LIN {X 0,Y 390.118,Z 490.981,A -85,B 0,C 180,E1 -11473.897,E2 -11473.897} C_VEL
LIN {X 0,Y 390.11,Z 491.016,A -85,B 0,C 180,E1 -11476.798,E2 -11476.798} C_VEL
LIN {X 0,Y 390.064,Z 491.01,A -85,B 0,C 180,E1 -11479.562,E2 -11479.562} C_VEL
LIN {X 0,Y 390.038,Z 491.022,A -85,B 0,C 180,E1 -11482.449,E2 -11482.449} C_VEL
LIN {X 0,Y 390.06,Z 491.021,A -85,B 0,C 180,E1 -11486.045,E2 -11486.045} C_VEL
LIN {X 0,Y 390.038,Z 491.013,A -85,B 0,C 180,E1 -11488.498,E2 -11488.498} C_VEL
LIN {X 0,Y 390.109,Z 491.015,A -85,B 0,C 180,E1 -11492.07,E2 -11492.07} C_VEL
LIN {X 0,Y 390.071,Z 491.003,A -85,B 0,C 180,E1 -11495.519,E2 -11495.519} C_VEL
LIN {X 0,Y 390.054,Z 491.022,A -85,B 0,C 180,E1 -11498.878,E2 -11498.878} C_VEL
LIN {X 0,Y 390.119,Z 490.998,A -85,B 0,C 180,E1 -11502.167,E2 -11502.167} C_VEL
LIN {X 0,Y 390.135,Z 491.009,A -85,B 0,C 180,E1 -11505.393,E2 -11505.393} C_VEL
LIN {X 0,Y 390.139,Z 490.999,A -85,B 0,C 180,E1 -11508.571,E2 -11508.571} C_VEL
LIN {X 0,Y 390.298,Z 490.981,A -85,B 0,C 180,E1 -11512.033,E2 -11512.033} C_VEL
LIN {X 0,Y 390.225,Z 490.997,A -85,B 0,C 180,E1 -11514.834,E2 -11514.834} C_VEL
LIN {X 0,Y 390.412,Z 490.954,A -85,B 0,C 180,E1 -11517.937,E2 -11517.937} C_VEL
LIN {X 0,Y 390.541,Z 490.951,A -85,B 0,C 180,E1 -11520,E2 -11520} C_VEL
LIN {X 0,Y 390.308,Z 490.984,A -85,B 0,C 180,E1 -11523.097,E2 -11523.097} C_VEL
LIN {X 0,Y 390.32,Z 490.966,A -85,B 0,C 180,E1 -11526.202,E2 -11526.202} C_VEL
LIN {X 0,Y 390.197,Z 491.003,A -85,B 0,C 180,E1 -11529.329,E2 -11529.329} C_VEL
LIN {X 0,Y 390.187,Z 490.982,A -85,B 0,C 180,E1 -11533.439,E2 -11533.439} C_VEL
LIN {X 0,Y 390.142,Z 491.01,A -85,B 0,C 180,E1 -11537.308,E2 -11537.308} C_VEL
LIN {X 0,Y 390.081,Z 491.003,A -85,B 0,C 180,E1 -11540.471,E2 -11540.471} C_VEL
LIN {X 0,Y 390.072,Z 491.023,A -85,B 0,C 180,E1 -11544.482,E2 -11544.482} C_VEL
LIN {X 0,Y 390.112,Z 491.001,A -85,B 0,C 180,E1 -11547.931,E2 -11547.931} C_VEL
LIN {X 0,Y 390.018,Z 491.022,A -85,B 0,C 180,E1 -11551.505,E2 -11551.505} C_VEL
LIN {X 0,Y 390.081,Z 491.019,A -85,B 0,C 180,E1 -11555.208,E2 -11555.208} C_VEL
LIN {X 0,Y 390.091,Z 491.019,A -85,B 0,C 180,E1 -11559.093,E2 -11559.093} C_VEL
LIN {X 0,Y 390.077,Z 491.015,A -85,B 0,C 180,E1 -11562.381,E2 -11562.381} C_VEL
LIN {X 0,Y 390.054,Z 491.005,A -85,B 0,C 180,E1 -11566.115,E2 -11566.115} C_VEL
LIN {X 0,Y 390.055,Z 491.022,A -85,B 0,C 180,E1 -11569.562,E2 -11569.562} C_VEL
LIN {X 0,Y 390.042,Z 490.971,A -85,B 0,C 180,E1 -11572.45,E2 -11572.45} C_VEL
LIN {X 0,Y 390.067,Z 491.009,A -85,B 0,C 180,E1 -11575.976,E2 -11575.976} C_VEL
LIN {X 0,Y 390.107,Z 491.228,A -85,B 0,C 180,E1 -11577.132,E2 -11577.132} C_VEL
LIN {X 0,Y 392.197,Z 500.873,A -85,B 0,C 180,E1 -11579.885,E2 -11579.885} C_VEL
LIN {X 0,Y 394.038,Z 510.309,A -85,B 0,C 180,E1 -11582.373,E2 -11582.373} C_VEL
LIN {X 0,Y 394.142,Z 513.122,A -85,B 0,C 180,E1 -11583.07,E2 -11583.07} C_VEL
LIN {X 0,Y 393.369,Z 521.493,A -85,B 0,C 180,E1 -11585.111,E2 -11585.111} C_VEL
LIN {X 0,Y 394.757,Z 528.148,A -85,B 0,C 180,E1 -11585.38,E2 -11585.38} C_VEL
LIN {X 0,Y 400.375,Z 555.374,A -85,B 0,C 180,E1 -11586.267,E2 -11586.267} C_VEL
LIN {X 0,Y 400.741,Z 558.243,A -85,B 0,C 180,E1 -11586.345,E2 -11586.345} C_VEL
LIN {X 0,Y 398.955,Z 657.044,A -85,B 0,C 180,E1 -11588.153,E2 -11588.153} C_VEL
LIN {X 0,Y 398.444,Z 667.994,A -85,B 0,C 180,E1 -11588.463,E2 -11588.463} C_VEL
LIN {X 0,Y 397.788,Z 678.984,A -85,B 0,C 180,E1 -11588.902,E2 -11588.902} C_VEL
LIN {X 0,Y 397.102,Z 688.994,A -85,B 0,C 180,E1 -11589.42,E2 -11589.42} C_VEL
LIN {X 0,Y 396.287,Z 698.786,A -85,B 0,C 180,E1 -11590.042,E2 -11590.042} C_VEL
LIN {X 0,Y 395.442,Z 708.675,A -85,B 0,C 180,E1 -11590.805,E2 -11590.805} C_VEL
LIN {X 0,Y 394.447,Z 718.401,A -85,B 0,C 180,E1 -11591.698,E2 -11591.698} C_VEL
LIN {X 0,Y 393.41,Z 727.821,A -85,B 0,C 180,E1 -11592.723,E2 -11592.723} C_VEL
LIN {X 0,Y 392.435,Z 736.845,A -85,B 0,C 180,E1 -11593.884,E2 -11593.884} C_VEL
LIN {X 0,Y 391.671,Z 743.822,A -85,B 0,C 180,E1 -11594.919,E2 -11594.919} C_VEL
LIN {X 0,Y 390.934,Z 750.826,A -85,B 0,C 180,E1 -11596.117,E2 -11596.117} C_VEL
LIN {X 0,Y 390.32,Z 757.827,A -85,B 0,C 180,E1 -11597.522,E2 -11597.522} C_VEL
LIN {X 0,Y 389.661,Z 764.367,A -85,B 0,C 180,E1 -11599.084,E2 -11599.084} C_VEL
LIN {X 0,Y 389.23,Z 769.8,A -85,B 0,C 180,E1 -11600.648,E2 -11600.648} C_VEL
LIN {X 0,Y 388.923,Z 774.244,A -85,B 0,C 180,E1 -11602.211,E2 -11602.211} C_VEL
LIN {X 0,Y 388.775,Z 777.942,A -85,B 0,C 180,E1 -11603.856,E2 -11603.856} C_VEL
LIN {X 0,Y 388.707,Z 779.727,A -85,B 0,C 180,E1 -11604.813,E2 -11604.813} C_VEL
LIN {X 0,Y 388.63,Z 782.408,A -85,B 0,C 180,E1 -11606.89,E2 -11606.89} C_VEL
LIN {X 0,Y 388.702,Z 783.698,A -85,B 0,C 180,E1 -11608.964,E2 -11608.964} C_VEL
LIN {X 0,Y 388.707,Z 783.95,A -85,B 0,C 180,E1 -11610,E2 -11610} C_VEL
LIN {X 0,Y 388.659,Z 783.225,A -85,B 0,C 180,E1 -11612.073,E2 -11612.073} C_VEL
LIN {X 0,Y 388.63,Z 782.408,A -85,B 0,C 180,E1 -11613.11,E2 -11613.11} C_VEL
LIN {X 0,Y 388.704,Z 779.727,A -85,B 0,C 180,E1 -11615.187,E2 -11615.187} C_VEL
LIN {X 0,Y 388.845,Z 776.773,A -85,B 0,C 180,E1 -11616.747,E2 -11616.747} C_VEL
LIN {X 0,Y 389.002,Z 772.946,A -85,B 0,C 180,E1 -11618.31,E2 -11618.31} C_VEL
LIN {X 0,Y 389.339,Z 768.184,A -85,B 0,C 180,E1 -11619.874,E2 -11619.874} C_VEL
LIN {X 0,Y 389.993,Z 761.241,A -85,B 0,C 180,E1 -11621.697,E2 -11621.697} C_VEL
LIN {X 0,Y 390.661,Z 754.026,A -85,B 0,C 180,E1 -11623.26,E2 -11623.26} C_VEL
LIN {X 0,Y 391.34,Z 746.947,A -85,B 0,C 180,E1 -11624.561,E2 -11624.561} C_VEL
LIN {X 0,Y 392.036,Z 740.483,A -85,B 0,C 180,E1 -11625.599,E2 -11625.599} C_VEL
LIN {X 0,Y 393.053,Z 731,A -85,B 0,C 180,E1 -11626.891,E2 -11626.891} C_VEL
LIN {X 0,Y 394.065,Z 722.123,A -85,B 0,C 180,E1 -11627.917,E2 -11627.917} C_VEL
LIN {X 0,Y 395.042,Z 713.07,A -85,B 0,C 180,E1 -11628.811,E2 -11628.811} C_VEL
LIN {X 0,Y 396.028,Z 702.261,A -85,B 0,C 180,E1 -11629.705,E2 -11629.705} C_VEL
LIN {X 0,Y 396.826,Z 692.523,A -85,B 0,C 180,E1 -11630.373,E2 -11630.373} C_VEL
LIN {X 0,Y 397.585,Z 681.704,A -85,B 0,C 180,E1 -11630.974,E2 -11630.974} C_VEL
LIN {X 0,Y 398.346,Z 669.818,A -85,B 0,C 180,E1 -11631.474,E2 -11631.474} C_VEL
LIN {X 0,Y 398.878,Z 658.403,A -85,B 0,C 180,E1 -11631.817,E2 -11631.817} C_VEL
LIN {X 0,Y 399.554,Z 628.292,A -85,B 0,C 180,E1 -11632.39,E2 -11632.39} C_VEL
LIN {X 0,Y 400.705,Z 557.213,A -85,B 0,C 180,E1 -11633.677,E2 -11633.677} C_VEL
LIN {X 0,Y 394.872,Z 528.424,A -85,B 0,C 180,E1 -11634.607,E2 -11634.607} C_VEL
LIN {X 0,Y 393.382,Z 521.582,A -85,B 0,C 180,E1 -11634.877,E2 -11634.877} C_VEL
LIN {X 0,Y 394.231,Z 512.042,A -85,B 0,C 180,E1 -11637.195,E2 -11637.195} C_VEL
LIN {X 0,Y 392.995,Z 504.589,A -85,B 0,C 180,E1 -11639.163,E2 -11639.163} C_VEL
LIN {X 0,Y 390.582,Z 493.387,A -85,B 0,C 180,E1 -11642.252,E2 -11642.252} C_VEL
LIN {X 0,Y 390.082,Z 491.039,A -85,B 0,C 180,E1 -11643.005,E2 -11643.005} C_VEL
LIN {X 0,Y 390.055,Z 490.963,A -85,B 0,C 180,E1 -11646.483,E2 -11646.483} C_VEL
LIN {X 0,Y 390.069,Z 491.006,A -85,B 0,C 180,E1 -11649.218,E2 -11649.218} C_VEL
LIN {X 0,Y 390.042,Z 491.009,A -85,B 0,C 180,E1 -11652.374,E2 -11652.374} C_VEL
LIN {X 0,Y 390.042,Z 491.021,A -85,B 0,C 180,E1 -11655.354,E2 -11655.354} C_VEL
LIN {X 0,Y 390.065,Z 491.014,A -85,B 0,C 180,E1 -11658.191,E2 -11658.191} C_VEL
LIN {X 0,Y 390.091,Z 491.018,A -85,B 0,C 180,E1 -11660.907,E2 -11660.907} C_VEL
LIN {X 0,Y 390.081,Z 491.019,A -85,B 0,C 180,E1 -11664.792,E2 -11664.792} C_VEL
LIN {X 0,Y 390.018,Z 491.022,A -85,B 0,C 180,E1 -11668.495,E2 -11668.495} C_VEL
LIN {X 0,Y 390.112,Z 491.001,A -85,B 0,C 180,E1 -11672.069,E2 -11672.069} C_VEL
LIN {X 0,Y 390.072,Z 491.023,A -85,B 0,C 180,E1 -11675.518,E2 -11675.518} C_VEL
LIN {X 0,Y 390.081,Z 491.003,A -85,B 0,C 180,E1 -11679.529,E2 -11679.529} C_VEL
LIN {X 0,Y 390.131,Z 491.015,A -85,B 0,C 180,E1 -11683.247,E2 -11683.247} C_VEL
LIN {X 0,Y 390.187,Z 490.982,A -85,B 0,C 180,E1 -11686.561,E2 -11686.561} C_VEL
LIN {X 0,Y 390.197,Z 491.003,A -85,B 0,C 180,E1 -11690.671,E2 -11690.671} C_VEL
LIN {X 0,Y 390.32,Z 490.966,A -85,B 0,C 180,E1 -11693.798,E2 -11693.798} C_VEL
LIN {X 0,Y 390.412,Z 490.976,A -85,B 0,C 180,E1 -11697.936,E2 -11697.936} C_VEL
LIN {X 0,Y 390.541,Z 490.951,A -85,B 0,C 180,E1 -11700,E2 -11700} C_VEL
LIN {X 0,Y 390.308,Z 490.97,A -85,B 0,C 180,E1 -11703.096,E2 -11703.096} C_VEL
LIN {X 0,Y 390.293,Z 490.989,A -85,B 0,C 180,E1 -11706.649,E2 -11706.649} C_VEL
LIN {X 0,Y 390.196,Z 490.986,A -85,B 0,C 180,E1 -11709.328,E2 -11709.328} C_VEL
LIN {X 0,Y 390.186,Z 491.008,A -85,B 0,C 180,E1 -11713.438,E2 -11713.438} C_VEL
LIN {X 0,Y 390.14,Z 490.994,A -85,B 0,C 180,E1 -11717.307,E2 -11717.307} C_VEL
LIN {X 0,Y 390.079,Z 491.017,A -85,B 0,C 180,E1 -11720.47,E2 -11720.47} C_VEL
LIN {X 0,Y 390.08,Z 491.008,A -85,B 0,C 180,E1 -11723.351,E2 -11723.351} C_VEL
LIN {X 0,Y 390.105,Z 491.013,A -85,B 0,C 180,E1 -11726.768,E2 -11726.768} C_VEL
LIN {X 0,Y 390.036,Z 491.009,A -85,B 0,C 180,E1 -11730.299,E2 -11730.299} C_VEL
LIN {X 0,Y 390.047,Z 491.021,A -85,B 0,C 180,E1 -11732.72,E2 -11732.72} C_VEL
LIN {X 0,Y 390.049,Z 491.013,A -85,B 0,C 180,E1 -11735.826,E2 -11735.826} C_VEL
LIN {X 0,Y 390.064,Z 491.022,A -85,B 0,C 180,E1 -11739.219,E2 -11739.219} C_VEL
LIN {X 0,Y 390.114,Z 491.015,A -85,B 0,C 180,E1 -11742.387,E2 -11742.387} C_VEL
LIN {X 0,Y 390.11,Z 490.994,A -85,B 0,C 180,E1 -11745.365,E2 -11745.365} C_VEL
LIN {X 0,Y 390.098,Z 490.993,A -85,B 0,C 180,E1 -11748.197,E2 -11748.197} C_VEL
LIN {X 0,Y 390.09,Z 491.018,A -85,B 0,C 180,E1 -11750.909,E2 -11750.909} C_VEL
LIN {X 0,Y 390.079,Z 491.013,A -85,B 0,C 180,E1 -11754.793,E2 -11754.793} C_VEL
LIN {X 0,Y 390.028,Z 491.03,A -85,B 0,C 180,E1 -11757.875,E2 -11757.875} C_VEL
LIN {X 0,Y 390.06,Z 491.023,A -85,B 0,C 180,E1 -11760.891,E2 -11760.891} C_VEL
LIN {X 0,Y 390.106,Z 491.018,A -85,B 0,C 180,E1 -11764.382,E2 -11764.382} C_VEL
LIN {X 0,Y 390.035,Z 491.028,A -85,B 0,C 180,E1 -11767.766,E2 -11767.766} C_VEL
LIN {X 0,Y 390.101,Z 491.019,A -85,B 0,C 180,E1 -11771.078,E2 -11771.078} C_VEL
LIN {X 0,Y 390.135,Z 491.015,A -85,B 0,C 180,E1 -11774.323,E2 -11774.323} C_VEL
LIN {X 0,Y 390.167,Z 491.011,A -85,B 0,C 180,E1 -11777.517,E2 -11777.517} C_VEL
LIN {X 0,Y 390.241,Z 491.299,A -85,B 0,C 180,E1 -11780.378,E2 -11780.378} C_VEL
LIN {X 0,Y 390.604,Z 492.537,A -85,B 0,C 180,E1 -11781.137,E2 -11781.137} C_VEL
LIN {X 0,Y 392.054,Z 494.823,A -85,B 0,C 180,E1 -11782.457,E2 -11782.457} C_VEL
LIN {X 0,Y 393.897,Z 496.346,A -85,B 0,C 180,E1 -11784.369,E2 -11784.369} C_VEL
LIN {X 0,Y 395.019,Z 496.962,A -85,B 0,C 180,E1 -11785.919,E2 -11785.919} C_VEL
LIN {X 0,Y 395.996,Z 497.339,A -85,B 0,C 180,E1 -11787.966,E2 -11787.966} C_VEL
LIN {X 0,Y 396.223,Z 497.592,A -85,B 0,C 180,E1 -11788.984,E2 -11788.984} C_VEL
LIN {X 0,Y 396.324,Z 497.476,A -85,B 0,C 180,E1 -11790,E2 -11790} C_VEL
LIN {X 0,Y 396.113,Z 497.471,A -85,B 0,C 180,E1 -11791.525,E2 -11791.525} C_VEL
LIN {X 0,Y 395.594,Z 497.134,A -85,B 0,C 180,E1 -11793.055,E2 -11793.055} C_VEL
LIN {X 0,Y 394.296,Z 496.586,A -85,B 0,C 180,E1 -11795.113,E2 -11795.113} C_VEL
LIN {X 0,Y 392.392,Z 495.186,A -85,B 0,C 180,E1 -11797.202,E2 -11797.202} C_VEL
LIN {X 0,Y 390.757,Z 492.871,A -85,B 0,C 180,E1 -11798.717,E2 -11798.717} C_VEL
LIN {X 0,Y 390.301,Z 491.64,A -85,B 0,C 180,E1 -11799.326,E2 -11799.326} C_VEL
LIN {X 0,Y 390.165,Z 491.041,A -85,B 0,C 180,E1 -11800.377,E2 -11800.377} C_VEL
LIN {X 0,Y 390.165,Z 491.011,A -85,B 0,C 180,E1 -11803.542,E2 -11803.542} C_VEL
LIN {X 0,Y 390.144,Z 491.014,A -85,B 0,C 180,E1 -11807.307,E2 -11807.307} C_VEL
LIN {X 0,Y 390.082,Z 491.022,A -85,B 0,C 180,E1 -11810.47,E2 -11810.47} C_VEL
LIN {X 0,Y 390.084,Z 491.021,A -85,B 0,C 180,E1 -11813.351,E2 -11813.351} C_VEL
LIN {X 0,Y 390.108,Z 491.018,A -85,B 0,C 180,E1 -11816.768,E2 -11816.768} C_VEL
LIN {X 0,Y 390.038,Z 491.028,A -85,B 0,C 180,E1 -11820.299,E2 -11820.299} C_VEL
LIN {X 0,Y 390.01,Z 491.028,A -85,B 0,C 180,E1 -11820.819,E2 -11820.819} C_VEL
LIN {X 0,Y 389.336,Z 491.114,A -85,B 0,C 180,E1 -11821.681,E2 -11821.681} C_VEL
LIN {X 0,Y 386.486,Z 491.468,A -85,B 0,C 180,E1 -11823.083,E2 -11823.083} C_VEL
LIN {X 0,Y 384.087,Z 491.769,A -85,B 0,C 180,E1 -11824.216,E2 -11824.216} C_VEL
LIN {X 0,Y 383.069,Z 491.887,A -85,B 0,C 180,E1 -11825.092,E2 -11825.092} C_VEL
LIN {X 0,Y 382.993,Z 491.887,A -85,B 0,C 180,E1 -11825.388,E2 -11825.388} C_VEL
LIN {X 0,Y 383.003,Z 491.896,A -85,B 0,C 180,E1 -11828.6,E2 -11828.6} C_VEL
LIN {X 0,Y 383.04,Z 491.882,A -85,B 0,C 180,E1 -11831.339,E2 -11831.339} C_VEL
LIN {X 0,Y 383.061,Z 491.865,A -85,B 0,C 180,E1 -11834.314,E2 -11834.314} C_VEL
LIN {X 0,Y 383.068,Z 491.892,A -85,B 0,C 180,E1 -11837.249,E2 -11837.249} C_VEL
LIN {X 0,Y 383.012,Z 491.898,A -85,B 0,C 180,E1 -11840.412,E2 -11840.412} C_VEL
LIN {X 0,Y 383.018,Z 491.888,A -85,B 0,C 180,E1 -11844.044,E2 -11844.044} C_VEL
LIN {X 0,Y 383.028,Z 491.897,A -85,B 0,C 180,E1 -11847.853,E2 -11847.853} C_VEL
LIN {X 0,Y 383.055,Z 491.891,A -85,B 0,C 180,E1 -11851.72,E2 -11851.72} C_VEL
LIN {X 0,Y 383.043,Z 491.879,A -85,B 0,C 180,E1 -11855.04,E2 -11855.04} C_VEL
LIN {X 0,Y 382.99,Z 491.904,A -85,B 0,C 180,E1 -11858.469,E2 -11858.469} C_VEL
LIN {X 0,Y 383.08,Z 491.877,A -85,B 0,C 180,E1 -11861.828,E2 -11861.828} C_VEL
LIN {X 0,Y 383.101,Z 491.886,A -85,B 0,C 180,E1 -11865.118,E2 -11865.118} C_VEL
LIN {X 0,Y 383.089,Z 491.88,A -85,B 0,C 180,E1 -11868.358,E2 -11868.358} C_VEL
LIN {X 0,Y 383.255,Z 491.858,A -85,B 0,C 180,E1 -11871.976,E2 -11871.976} C_VEL
LIN {X 0,Y 383.197,Z 491.873,A -85,B 0,C 180,E1 -11874.739,E2 -11874.739} C_VEL
LIN {X 0,Y 383.38,Z 491.829,A -85,B 0,C 180,E1 -11877.899,E2 -11877.899} C_VEL
LIN {X 0,Y 383.511,Z 491.827,A -85,B 0,C 180,E1 -11880,E2 -11880} C_VEL
LIN {X 0,Y 383.244,Z 491.863,A -85,B 0,C 180,E1 -11883.154,E2 -11883.154} C_VEL
LIN {X 0,Y 383.277,Z 491.844,A -85,B 0,C 180,E1 -11886.317,E2 -11886.317} C_VEL
LIN {X 0,Y 383.144,Z 491.881,A -85,B 0,C 180,E1 -11889.503,E2 -11889.503} C_VEL
LIN {X 0,Y 383.118,Z 491.862,A -85,B 0,C 180,E1 -11893.537,E2 -11893.537} C_VEL
LIN {X 0,Y 383.088,Z 491.888,A -85,B 0,C 180,E1 -11897.455,E2 -11897.455} C_VEL
LIN {X 0,Y 383.022,Z 491.881,A -85,B 0,C 180,E1 -11900.647,E2 -11900.647} C_VEL
LIN {X 0,Y 383.02,Z 491.897,A -85,B 0,C 180,E1 -11903.809,E2 -11903.809} C_VEL
LIN {X 0,Y 383.074,Z 491.884,A -85,B 0,C 180,E1 -11906.124,E2 -11906.124} C_VEL
LIN {X 0,Y 382.986,Z 491.901,A -85,B 0,C 180,E1 -11909.701,E2 -11909.701} C_VEL
LIN {X 0,Y 382.998,Z 491.89,A -85,B 0,C 180,E1 -11913.402,E2 -11913.402} C_VEL
LIN {X 0,Y 383.029,Z 491.898,A -85,B 0,C 180,E1 -11916.166,E2 -11916.166} C_VEL
LIN {X 0,Y 383.016,Z 491.9,A -85,B 0,C 180,E1 -11919.958,E2 -11919.958} C_VEL
LIN {X 0,Y 383.029,Z 491.896,A -85,B 0,C 180,E1 -11922.784,E2 -11922.784} C_VEL
LIN {X 0,Y 382.996,Z 491.887,A -85,B 0,C 180,E1 -11925.79,E2 -11925.79} C_VEL
LIN {X 0,Y 382.987,Z 491.902,A -85,B 0,C 180,E1 -11928.797,E2 -11928.797} C_VEL
LIN {X 0,Y 382.998,Z 491.852,A -85,B 0,C 180,E1 -11932.097,E2 -11932.097} C_VEL
LIN {X 0,Y 383.017,Z 491.864,A -85,B 0,C 180,E1 -11935.333,E2 -11935.333} C_VEL
LIN {X 0,Y 383.077,Z 492.078,A -85,B 0,C 180,E1 -11936.728,E2 -11936.728} C_VEL
LIN {X 0,Y 385.189,Z 501.84,A -85,B 0,C 180,E1 -11939.582,E2 -11939.582} C_VEL
LIN {X 0,Y 387.187,Z 512.271,A -85,B 0,C 180,E1 -11942.383,E2 -11942.383} C_VEL
LIN {X 0,Y 386.939,Z 516.944,A -85,B 0,C 180,E1 -11943.578,E2 -11943.578} C_VEL
LIN {X 0,Y 386.564,Z 521.303,A -85,B 0,C 180,E1 -11944.645,E2 -11944.645} C_VEL
LIN {X 0,Y 388.306,Z 529.362,A -85,B 0,C 180,E1 -11944.971,E2 -11944.971} C_VEL
LIN {X 0,Y 394.047,Z 557.41,A -85,B 0,C 180,E1 -11945.906,E2 -11945.906} C_VEL
LIN {X 0,Y 393.732,Z 585.51,A -85,B 0,C 180,E1 -11946.433,E2 -11946.433} C_VEL
LIN {X 0,Y 392.374,Z 656.846,A -85,B 0,C 180,E1 -11947.767,E2 -11947.767} C_VEL
LIN {X 0,Y 391.856,Z 667.796,A -85,B 0,C 180,E1 -11948.083,E2 -11948.083} C_VEL
LIN {X 0,Y 391.176,Z 678.786,A -85,B 0,C 180,E1 -11948.527,E2 -11948.527} C_VEL
LIN {X 0,Y 390.448,Z 688.583,A -85,B 0,C 180,E1 -11949.039,E2 -11949.039} C_VEL
LIN {X 0,Y 389.575,Z 698.907,A -85,B 0,C 180,E1 -11949.708,E2 -11949.708} C_VEL
LIN {X 0,Y 388.729,Z 708.52,A -85,B 0,C 180,E1 -11950.464,E2 -11950.464} C_VEL
LIN {X 0,Y 387.702,Z 718.202,A -85,B 0,C 180,E1 -11951.368,E2 -11951.368} C_VEL
LIN {X 0,Y 386.601,Z 727.622,A -85,B 0,C 180,E1 -11952.409,E2 -11952.409} C_VEL
LIN {X 0,Y 385.56,Z 736.645,A -85,B 0,C 180,E1 -11953.589,E2 -11953.589} C_VEL
LIN {X 0,Y 384.758,Z 743.622,A -85,B 0,C 180,E1 -11954.642,E2 -11954.642} C_VEL
LIN {X 0,Y 383.905,Z 751.284,A -85,B 0,C 180,E1 -11955.99,E2 -11955.99} C_VEL
LIN {X 0,Y 383.234,Z 758.766,A -85,B 0,C 180,E1 -11957.557,E2 -11957.557} C_VEL
LIN {X 0,Y 382.637,Z 764.167,A -85,B 0,C 180,E1 -11958.881,E2 -11958.881} C_VEL
LIN {X 0,Y 382.165,Z 769.6,A -85,B 0,C 180,E1 -11960.473,E2 -11960.473} C_VEL
LIN {X 0,Y 381.851,Z 774.045,A -85,B 0,C 180,E1 -11962.066,E2 -11962.066} C_VEL
LIN {X 0,Y 381.71,Z 777.59,A -85,B 0,C 180,E1 -11963.658,E2 -11963.658} C_VEL
LIN {X 0,Y 381.616,Z 779.528,A -85,B 0,C 180,E1 -11964.717,E2 -11964.717} C_VEL
LIN {X 0,Y 381.541,Z 782.21,A -85,B 0,C 180,E1 -11966.832,E2 -11966.832} C_VEL
LIN {X 0,Y 381.616,Z 783.5,A -85,B 0,C 180,E1 -11968.945,E2 -11968.945} C_VEL
LIN {X 0,Y 381.638,Z 783.753,A -85,B 0,C 180,E1 -11970,E2 -11970} C_VEL
LIN {X 0,Y 381.558,Z 783.027,A -85,B 0,C 180,E1 -11972.111,E2 -11972.111} C_VEL
LIN {X 0,Y 381.541,Z 782.21,A -85,B 0,C 180,E1 -11973.168,E2 -11973.168} C_VEL
LIN {X 0,Y 381.615,Z 779.528,A -85,B 0,C 180,E1 -11975.283,E2 -11975.283} C_VEL
LIN {X 0,Y 381.757,Z 776.574,A -85,B 0,C 180,E1 -11976.872,E2 -11976.872} C_VEL
LIN {X 0,Y 381.95,Z 772.747,A -85,B 0,C 180,E1 -11978.465,E2 -11978.465} C_VEL
LIN {X 0,Y 382.301,Z 767.985,A -85,B 0,C 180,E1 -11980.058,E2 -11980.058} C_VEL
LIN {X 0,Y 382.974,Z 761.041,A -85,B 0,C 180,E1 -11981.914,E2 -11981.914} C_VEL
LIN {X 0,Y 383.555,Z 755.164,A -85,B 0,C 180,E1 -11983.24,E2 -11983.24} C_VEL
LIN {X 0,Y 384.429,Z 746.748,A -85,B 0,C 180,E1 -11984.829,E2 -11984.829} C_VEL
LIN {X 0,Y 385.167,Z 740.284,A -85,B 0,C 180,E1 -11985.884,E2 -11985.884} C_VEL
LIN {X 0,Y 386.213,Z 730.801,A -85,B 0,C 180,E1 -11987.199,E2 -11987.199} C_VEL
LIN {X 0,Y 387.287,Z 721.924,A -85,B 0,C 180,E1 -11988.242,E2 -11988.242} C_VEL
LIN {X 0,Y 388.305,Z 712.871,A -85,B 0,C 180,E1 -11989.15,E2 -11989.15} C_VEL
LIN {X 0,Y 389.329,Z 702.062,A -85,B 0,C 180,E1 -11990.058,E2 -11990.058} C_VEL
LIN {X 0,Y 390.264,Z 691.158,A -85,B 0,C 180,E1 -11990.806,E2 -11990.806} C_VEL
LIN {X 0,Y 391.058,Z 680.146,A -85,B 0,C 180,E1 -11991.41,E2 -11991.41} C_VEL
LIN {X 0,Y 391.808,Z 668.708,A -85,B 0,C 180,E1 -11991.885,E2 -11991.885} C_VEL
LIN {X 0,Y 392.303,Z 658.205,A -85,B 0,C 180,E1 -11992.202,E2 -11992.202} C_VEL
LIN {X 0,Y 393.006,Z 628.094,A -85,B 0,C 180,E1 -11992.784,E2 -11992.784} C_VEL
LIN {X 0,Y 394.133,Z 557.774,A -85,B 0,C 180,E1 -11994.082,E2 -11994.082} C_VEL
LIN {X 0,Y 388.314,Z 529.209,A -85,B 0,C 180,E1 -11995.032,E2 -11995.032} C_VEL
LIN {X 0,Y 386.58,Z 521.374,A -85,B 0,C 180,E1 -11995.345,E2 -11995.345} C_VEL
LIN {X 0,Y 387.295,Z 513.75,A -85,B 0,C 180,E1 -11997.23,E2 -11997.23} C_VEL
LIN {X 0,Y 386.212,Z 506.655,A -85,B 0,C 180,E1 -11999.135,E2 -11999.135} C_VEL
LIN {X 0,Y 383.975,Z 496.243,A -85,B 0,C 180,E1 -12002.058,E2 -12002.058} C_VEL
LIN {X 0,Y 383.069,Z 491.935,A -85,B 0,C 180,E1 -12003.363,E2 -12003.363} C_VEL
LIN {X 0,Y 383.03,Z 491.837,A -85,B 0,C 180,E1 -12006.164,E2 -12006.164} C_VEL
LIN {X 0,Y 383.007,Z 491.9,A -85,B 0,C 180,E1 -12009.957,E2 -12009.957} C_VEL
LIN {X 0,Y 383.003,Z 491.881,A -85,B 0,C 180,E1 -12012.778,E2 -12012.778} C_VEL
LIN {X 0,Y 382.995,Z 491.903,A -85,B 0,C 180,E1 -12015.788,E2 -12015.788} C_VEL
LIN {X 0,Y 383.011,Z 491.894,A -85,B 0,C 180,E1 -12018.79,E2 -12018.79} C_VEL
LIN {X 0,Y 382.999,Z 491.892,A -85,B 0,C 180,E1 -12022.095,E2 -12022.095} C_VEL
LIN {X 0,Y 383.014,Z 491.896,A -85,B 0,C 180,E1 -12025.331,E2 -12025.331} C_VEL
LIN {X 0,Y 382.977,Z 491.903,A -85,B 0,C 180,E1 -12029.081,E2 -12029.081} C_VEL
LIN {X 0,Y 383.051,Z 491.879,A -85,B 0,C 180,E1 -12032.697,E2 -12032.697} C_VEL
LIN {X 0,Y 383.045,Z 491.892,A -85,B 0,C 180,E1 -12035.039,E2 -12035.039} C_VEL
LIN {X 0,Y 382.985,Z 491.89,A -85,B 0,C 180,E1 -12038.468,E2 -12038.468} C_VEL
LIN {X 0,Y 383.082,Z 491.891,A -85,B 0,C 180,E1 -12041.827,E2 -12041.827} C_VEL
LIN {X 0,Y 383.102,Z 491.877,A -85,B 0,C 180,E1 -12045.118,E2 -12045.118} C_VEL
LIN {X 0,Y 383.09,Z 491.883,A -85,B 0,C 180,E1 -12048.357,E2 -12048.357} C_VEL
LIN {X 0,Y 383.257,Z 491.862,A -85,B 0,C 180,E1 -12051.974,E2 -12051.974} C_VEL
LIN {X 0,Y 383.191,Z 491.853,A -85,B 0,C 180,E1 -12054.738,E2 -12054.738} C_VEL
LIN {X 0,Y 383.38,Z 491.852,A -85,B 0,C 180,E1 -12057.898,E2 -12057.898} C_VEL
LIN {X 0,Y 383.511,Z 491.827,A -85,B 0,C 180,E1 -12060,E2 -12060} C_VEL
LIN {X 0,Y 383.244,Z 491.85,A -85,B 0,C 180,E1 -12063.153,E2 -12063.153} C_VEL
LIN {X 0,Y 383.252,Z 491.865,A -85,B 0,C 180,E1 -12066.641,E2 -12066.641} C_VEL
LIN {X 0,Y 383.143,Z 491.863,A -85,B 0,C 180,E1 -12069.502,E2 -12069.502} C_VEL
LIN {X 0,Y 383.117,Z 491.889,A -85,B 0,C 180,E1 -12073.536,E2 -12073.536} C_VEL
LIN {X 0,Y 383.086,Z 491.872,A -85,B 0,C 180,E1 -12077.454,E2 -12077.454} C_VEL
LIN {X 0,Y 383.022,Z 491.896,A -85,B 0,C 180,E1 -12080.648,E2 -12080.648} C_VEL
LIN {X 0,Y 383.024,Z 491.882,A -85,B 0,C 180,E1 -12083.807,E2 -12083.807} C_VEL
LIN {X 0,Y 383.071,Z 491.891,A -85,B 0,C 180,E1 -12086.123,E2 -12086.123} C_VEL
LIN {X 0,Y 383.041,Z 491.892,A -85,B 0,C 180,E1 -12088.492,E2 -12088.492} C_VEL
LIN {X 0,Y 383,Z 491.899,A -85,B 0,C 180,E1 -12092.427,E2 -12092.427} C_VEL
LIN {X 0,Y 383.018,Z 491.888,A -85,B 0,C 180,E1 -12095.956,E2 -12095.956} C_VEL
LIN {X 0,Y 383.012,Z 491.898,A -85,B 0,C 180,E1 -12099.588,E2 -12099.588} C_VEL
LIN {X 0,Y 383.058,Z 491.894,A -85,B 0,C 180,E1 -12102.788,E2 -12102.788} C_VEL
LIN {X 0,Y 383.062,Z 491.863,A -85,B 0,C 180,E1 -12105.8,E2 -12105.8} C_VEL
LIN {X 0,Y 383.038,Z 491.886,A -85,B 0,C 180,E1 -12108.786,E2 -12108.786} C_VEL
LIN {X 0,Y 382.997,Z 491.886,A -85,B 0,C 180,E1 -12112.096,E2 -12112.096} C_VEL
LIN {X 0,Y 383.012,Z 491.898,A -85,B 0,C 180,E1 -12115.332,E2 -12115.332} C_VEL
LIN {X 0,Y 382.981,Z 491.905,A -85,B 0,C 180,E1 -12119.082,E2 -12119.082} C_VEL
LIN {X 0,Y 383.051,Z 491.897,A -85,B 0,C 180,E1 -12122.698,E2 -12122.698} C_VEL
LIN {X 0,Y 383.028,Z 491.9,A -85,B 0,C 180,E1 -12126.193,E2 -12126.193} C_VEL
LIN {X 0,Y 383.05,Z 491.897,A -85,B 0,C 180,E1 -12129.599,E2 -12129.599} C_VEL
LIN {X 0,Y 383.1,Z 491.892,A -85,B 0,C 180,E1 -12132.932,E2 -12132.932} C_VEL
LIN {X 0,Y 383.196,Z 492.132,A -85,B 0,C 180,E1 -12136.59,E2 -12136.59} C_VEL
LIN {X 0,Y 383.443,Z 493.257,A -85,B 0,C 180,E1 -12137.11,E2 -12137.11} C_VEL
LIN {X 0,Y 384.779,Z 495.64,A -85,B 0,C 180,E1 -12137.942,E2 -12137.942} C_VEL
LIN {X 0,Y 386.586,Z 497.173,A -85,B 0,C 180,E1 -12139.019,E2 -12139.019} C_VEL
LIN {X 0,Y 389.002,Z 498.608,A -85,B 0,C 180,E1 -12140.577,E2 -12140.577} C_VEL
LIN {X 0,Y 390.336,Z 500.879,A -85,B 0,C 180,E1 -12141.719,E2 -12141.719} C_VEL
LIN {X 0,Y 391.901,Z 502.624,A -85,B 0,C 180,E1 -12143.177,E2 -12143.177} C_VEL
LIN {X 0,Y 393.414,Z 503.635,A -85,B 0,C 180,E1 -12144.876,E2 -12144.876} C_VEL
LIN {X 0,Y 394.726,Z 504.158,A -85,B 0,C 180,E1 -12146.938,E2 -12146.938} C_VEL
LIN {X 0,Y 395.358,Z 504.638,A -85,B 0,C 180,E1 -12148.981,E2 -12148.981} C_VEL
LIN {X 0,Y 395.358,Z 504.639,A -85,B 0,C 180,E1 -12151.019,E2 -12151.019} C_VEL
LIN {X 0,Y 394.726,Z 504.155,A -85,B 0,C 180,E1 -12153.062,E2 -12153.062} C_VEL
LIN {X 0,Y 393.418,Z 503.612,A -85,B 0,C 180,E1 -12155.124,E2 -12155.124} C_VEL
LIN {X 0,Y 391.495,Z 502.25,A -85,B 0,C 180,E1 -12157.219,E2 -12157.219} C_VEL
LIN {X 0,Y 389.779,Z 500.121,A -85,B 0,C 180,E1 -12158.752,E2 -12158.752} C_VEL
LIN {X 0,Y 388.706,Z 498.318,A -85,B 0,C 180,E1 -12159.627,E2 -12159.627} C_VEL
LIN {X 0,Y 385.613,Z 496.448,A -85,B 0,C 180,E1 -12161.565,E2 -12161.565} C_VEL
LIN {X 0,Y 384.062,Z 494.607,A -85,B 0,C 180,E1 -12162.483,E2 -12162.483} C_VEL
LIN {X 0,Y 383.247,Z 492.572,A -85,B 0,C 180,E1 -12163.135,E2 -12163.135} C_VEL
LIN {X 0,Y 383.122,Z 491.933,A -85,B 0,C 180,E1 -12163.796,E2 -12163.796} C_VEL
LIN {X 0,Y 383.09,Z 491.892,A -85,B 0,C 180,E1 -12167.454,E2 -12167.454} C_VEL
LIN {X 0,Y 383.024,Z 491.902,A -85,B 0,C 180,E1 -12170.647,E2 -12170.647} C_VEL
LIN {X 0,Y 383.028,Z 491.9,A -85,B 0,C 180,E1 -12173.807,E2 -12173.807} C_VEL
LIN {X 0,Y 383.051,Z 491.897,A -85,B 0,C 180,E1 -12177.302,E2 -12177.302} C_VEL
LIN {X 0,Y 382.981,Z 491.905,A -85,B 0,C 180,E1 -12180.918,E2 -12180.918} C_VEL
LIN {X 0,Y 383.012,Z 491.898,A -85,B 0,C 180,E1 -12184.668,E2 -12184.668} C_VEL
LIN {X 0,Y 382.993,Z 491.887,A -85,B 0,C 180,E1 -12185.388,E2 -12185.388} C_VEL
LIN {X 0,Y 382.35,Z 491.964,A -85,B 0,C 180,E1 -12186.266,E2 -12186.266} C_VEL
LIN {X 0,Y 379.533,Z 492.33,A -85,B 0,C 180,E1 -12187.694,E2 -12187.694} C_VEL
LIN {X 0,Y 377.128,Z 492.641,A -85,B 0,C 180,E1 -12188.848,E2 -12188.848} C_VEL
LIN {X 0,Y 376.082,Z 492.77,A -85,B 0,C 180,E1 -12189.74,E2 -12189.74} C_VEL
LIN {X 0,Y 375.99,Z 492.777,A -85,B 0,C 180,E1 -12190.043,E2 -12190.043} C_VEL
LIN {X 0,Y 375.991,Z 492.737,A -85,B 0,C 180,E1 -12193.756,E2 -12193.756} C_VEL
LIN {X 0,Y 375.992,Z 492.775,A -85,B 0,C 180,E1 -12196.8,E2 -12196.8} C_VEL
LIN {X 0,Y 375.988,Z 492.767,A -85,B 0,C 180,E1 -12200.028,E2 -12200.028} C_VEL
LIN {X 0,Y 375.957,Z 492.769,A -85,B 0,C 180,E1 -12203.495,E2 -12203.495} C_VEL
LIN {X 0,Y 375.953,Z 492.777,A -85,B 0,C 180,E1 -12205.889,E2 -12205.889} C_VEL
LIN {X 0,Y 375.961,Z 492.761,A -85,B 0,C 180,E1 -12209.688,E2 -12209.688} C_VEL
LIN {X 0,Y 375.994,Z 492.774,A -85,B 0,C 180,E1 -12212.142,E2 -12212.142} C_VEL
LIN {X 0,Y 375.997,Z 492.761,A -85,B 0,C 180,E1 -12214.539,E2 -12214.539} C_VEL
LIN {X 0,Y 375.959,Z 492.775,A -85,B 0,C 180,E1 -12218.046,E2 -12218.046} C_VEL
LIN {X 0,Y 376.015,Z 492.76,A -85,B 0,C 180,E1 -12221.474,E2 -12221.474} C_VEL
LIN {X 0,Y 376.049,Z 492.766,A -85,B 0,C 180,E1 -12224.833,E2 -12224.833} C_VEL
LIN {X 0,Y 376.041,Z 492.761,A -85,B 0,C 180,E1 -12228.137,E2 -12228.137} C_VEL
LIN {X 0,Y 376.211,Z 492.735,A -85,B 0,C 180,E1 -12231.919,E2 -12231.919} C_VEL
LIN {X 0,Y 376.169,Z 492.75,A -85,B 0,C 180,E1 -12234.64,E2 -12234.64} C_VEL
LIN {X 0,Y 376.346,Z 492.704,A -85,B 0,C 180,E1 -12237.86,E2 -12237.86} C_VEL
LIN {X 0,Y 376.48,Z 492.702,A -85,B 0,C 180,E1 -12240.001,E2 -12240.001} C_VEL
LIN {X 0,Y 376.183,Z 492.743,A -85,B 0,C 180,E1 -12243.213,E2 -12243.213} C_VEL
LIN {X 0,Y 376.235,Z 492.721,A -85,B 0,C 180,E1 -12246.436,E2 -12246.436} C_VEL
LIN {X 0,Y 376.111,Z 492.758,A -85,B 0,C 180,E1 -12249.682,E2 -12249.682} C_VEL
LIN {X 0,Y 376.082,Z 492.738,A -85,B 0,C 180,E1 -12253.658,E2 -12253.658} C_VEL
LIN {X 0,Y 376.037,Z 492.766,A -85,B 0,C 180,E1 -12257.608,E2 -12257.608} C_VEL
LIN {X 0,Y 375.972,Z 492.759,A -85,B 0,C 180,E1 -12260.833,E2 -12260.833} C_VEL
LIN {X 0,Y 375.984,Z 492.776,A -85,B 0,C 180,E1 -12264.283,E2 -12264.283} C_VEL
LIN {X 0,Y 376.014,Z 492.757,A -85,B 0,C 180,E1 -12266.653,E2 -12266.653} C_VEL
LIN {X 0,Y 375.959,Z 492.779,A -85,B 0,C 180,E1 -12270.314,E2 -12270.314} C_VEL
LIN {X 0,Y 375.955,Z 492.77,A -85,B 0,C 180,E1 -12274.112,E2 -12274.112} C_VEL
LIN {X 0,Y 375.951,Z 492.776,A -85,B 0,C 180,E1 -12276.742,E2 -12276.742} C_VEL
LIN {X 0,Y 375.994,Z 492.774,A -85,B 0,C 180,E1 -12279.973,E2 -12279.973} C_VEL
LIN {X 0,Y 375.936,Z 492.782,A -85,B 0,C 180,E1 -12283.765,E2 -12283.765} C_VEL
LIN {X 0,Y 375.932,Z 492.76,A -85,B 0,C 180,E1 -12286.812,E2 -12286.812} C_VEL
LIN {X 0,Y 375.961,Z 492.766,A -85,B 0,C 180,E1 -12290.538,E2 -12290.538} C_VEL
LIN {X 0,Y 375.962,Z 492.714,A -85,B 0,C 180,E1 -12293.496,E2 -12293.496} C_VEL
LIN {X 0,Y 376.015,Z 492.918,A -85,B 0,C 180,E1 -12296.299,E2 -12296.299} C_VEL
LIN {X 0,Y 377.84,Z 501.257,A -85,B 0,C 180,E1 -12298.829,E2 -12298.829} C_VEL
LIN {X 0,Y 380.078,Z 512.248,A -85,B 0,C 180,E1 -12301.868,E2 -12301.868} C_VEL
LIN {X 0,Y 380.347,Z 515.117,A -85,B 0,C 180,E1 -12302.652,E2 -12302.652} C_VEL
LIN {X 0,Y 379.777,Z 521.222,A -85,B 0,C 180,E1 -12304.173,E2 -12304.173} C_VEL
LIN {X 0,Y 384.822,Z 544.293,A -85,B 0,C 180,E1 -12305.032,E2 -12305.032} C_VEL
LIN {X 0,Y 387.733,Z 559.553,A -85,B 0,C 180,E1 -12305.534,E2 -12305.534} C_VEL
LIN {X 0,Y 385.84,Z 655.308,A -85,B 0,C 180,E1 -12307.335,E2 -12307.335} C_VEL
LIN {X 0,Y 385.325,Z 666.686,A -85,B 0,C 180,E1 -12307.656,E2 -12307.656} C_VEL
LIN {X 0,Y 384.678,Z 677.228,A -85,B 0,C 180,E1 -12308.076,E2 -12308.076} C_VEL
LIN {X 0,Y 383.895,Z 687.416,A -85,B 0,C 180,E1 -12308.6,E2 -12308.6} C_VEL
LIN {X 0,Y 383.08,Z 697.285,A -85,B 0,C 180,E1 -12309.234,E2 -12309.234} C_VEL
LIN {X 0,Y 381.979,Z 708.796,A -85,B 0,C 180,E1 -12310.15,E2 -12310.15} C_VEL
LIN {X 0,Y 380.968,Z 718.004,A -85,B 0,C 180,E1 -12311.026,E2 -12311.026} C_VEL
LIN {X 0,Y 379.77,Z 727.422,A -85,B 0,C 180,E1 -12312.082,E2 -12312.082} C_VEL
LIN {X 0,Y 378.723,Z 736.446,A -85,B 0,C 180,E1 -12313.284,E2 -12313.284} C_VEL
LIN {X 0,Y 377.856,Z 743.422,A -85,B 0,C 180,E1 -12314.354,E2 -12314.354} C_VEL
LIN {X 0,Y 376.878,Z 751.745,A -85,B 0,C 180,E1 -12315.859,E2 -12315.859} C_VEL
LIN {X 0,Y 376.243,Z 758.566,A -85,B 0,C 180,E1 -12317.322,E2 -12317.322} C_VEL
LIN {X 0,Y 375.625,Z 763.968,A -85,B 0,C 180,E1 -12318.67,E2 -12318.67} C_VEL
LIN {X 0,Y 375.117,Z 769.401,A -85,B 0,C 180,E1 -12320.293,E2 -12320.293} C_VEL
LIN {X 0,Y 374.801,Z 773.846,A -85,B 0,C 180,E1 -12321.916,E2 -12321.916} C_VEL
LIN {X 0,Y 374.628,Z 777.391,A -85,B 0,C 180,E1 -12323.537,E2 -12323.537} C_VEL
LIN {X 0,Y 374.53,Z 779.33,A -85,B 0,C 180,E1 -12324.616,E2 -12324.616} C_VEL
LIN {X 0,Y 374.455,Z 782.012,A -85,B 0,C 180,E1 -12326.772,E2 -12326.772} C_VEL
LIN {X 0,Y 374.516,Z 783.302,A -85,B 0,C 180,E1 -12328.925,E2 -12328.925} C_VEL
LIN {X 0,Y 374.553,Z 783.555,A -85,B 0,C 180,E1 -12330,E2 -12330} C_VEL
LIN {X 0,Y 374.457,Z 782.828,A -85,B 0,C 180,E1 -12332.151,E2 -12332.151} C_VEL
LIN {X 0,Y 374.455,Z 782.012,A -85,B 0,C 180,E1 -12333.228,E2 -12333.228} C_VEL
LIN {X 0,Y 374.53,Z 779.33,A -85,B 0,C 180,E1 -12335.384,E2 -12335.384} C_VEL
LIN {X 0,Y 374.677,Z 776.375,A -85,B 0,C 180,E1 -12337.003,E2 -12337.003} C_VEL
LIN {X 0,Y 374.878,Z 772.548,A -85,B 0,C 180,E1 -12338.626,E2 -12338.626} C_VEL
LIN {X 0,Y 375.248,Z 767.785,A -85,B 0,C 180,E1 -12340.249,E2 -12340.249} C_VEL
LIN {X 0,Y 375.984,Z 760.842,A -85,B 0,C 180,E1 -12342.139,E2 -12342.139} C_VEL
LIN {X 0,Y 376.61,Z 754.965,A -85,B 0,C 180,E1 -12343.489,E2 -12343.489} C_VEL
LIN {X 0,Y 377.338,Z 748.112,A -85,B 0,C 180,E1 -12344.838,E2 -12344.838} C_VEL
LIN {X 0,Y 378.282,Z 740.085,A -85,B 0,C 180,E1 -12346.181,E2 -12346.181} C_VEL
LIN {X 0,Y 379.367,Z 730.601,A -85,B 0,C 180,E1 -12347.52,E2 -12347.52} C_VEL
LIN {X 0,Y 380.508,Z 721.724,A -85,B 0,C 180,E1 -12348.578,E2 -12348.578} C_VEL
LIN {X 0,Y 381.685,Z 711.424,A -85,B 0,C 180,E1 -12349.614,E2 -12349.614} C_VEL
LIN {X 0,Y 382.642,Z 701.864,A -85,B 0,C 180,E1 -12350.424,E2 -12350.424} C_VEL
LIN {X 0,Y 383.626,Z 690.96,A -85,B 0,C 180,E1 -12351.183,E2 -12351.183} C_VEL
LIN {X 0,Y 384.445,Z 679.948,A -85,B 0,C 180,E1 -12351.797,E2 -12351.797} C_VEL
LIN {X 0,Y 385.189,Z 669.422,A -85,B 0,C 180,E1 -12352.246,E2 -12352.246} C_VEL
LIN {X 0,Y 385.743,Z 658.007,A -85,B 0,C 180,E1 -12352.601,E2 -12352.601} C_VEL
LIN {X 0,Y 386.48,Z 627.896,A -85,B 0,C 180,E1 -12353.191,E2 -12353.191} C_VEL
LIN {X 0,Y 387.65,Z 558.758,A -85,B 0,C 180,E1 -12354.487,E2 -12354.487} C_VEL
LIN {X 0,Y 382.041,Z 531.207,A -85,B 0,C 180,E1 -12355.427,E2 -12355.427} C_VEL
LIN {X 0,Y 379.807,Z 521.353,A -85,B 0,C 180,E1 -12355.813,E2 -12355.813} C_VEL
LIN {X 0,Y 379.969,Z 518.94,A -85,B 0,C 180,E1 -12356.353,E2 -12356.353} C_VEL
LIN {X 0,Y 380.357,Z 514.5,A -85,B 0,C 180,E1 -12357.511,E2 -12357.511} C_VEL
LIN {X 0,Y 379.019,Z 506.787,A -85,B 0,C 180,E1 -12359.65,E2 -12359.65} C_VEL
LIN {X 0,Y 376.598,Z 495.581,A -85,B 0,C 180,E1 -12362.883,E2 -12362.883} C_VEL
LIN {X 0,Y 376.016,Z 492.796,A -85,B 0,C 180,E1 -12363.782,E2 -12363.782} C_VEL
LIN {X 0,Y 375.952,Z 492.716,A -85,B 0,C 180,E1 -12366.74,E2 -12366.74} C_VEL
LIN {X 0,Y 375.987,Z 492.774,A -85,B 0,C 180,E1 -12369.97,E2 -12369.97} C_VEL
LIN {X 0,Y 375.928,Z 492.761,A -85,B 0,C 180,E1 -12373.765,E2 -12373.765} C_VEL
LIN {X 0,Y 375.957,Z 492.772,A -85,B 0,C 180,E1 -12377.703,E2 -12377.703} C_VEL
LIN {X 0,Y 375.965,Z 492.777,A -85,B 0,C 180,E1 -12380.537,E2 -12380.537} C_VEL
LIN {X 0,Y 375.961,Z 492.778,A -85,B 0,C 180,E1 -12383.494,E2 -12383.494} C_VEL
LIN {X 0,Y 375.955,Z 492.77,A -85,B 0,C 180,E1 -12385.888,E2 -12385.888} C_VEL
LIN {X 0,Y 375.959,Z 492.779,A -85,B 0,C 180,E1 -12389.686,E2 -12389.686} C_VEL
LIN {X 0,Y 376.014,Z 492.757,A -85,B 0,C 180,E1 -12393.347,E2 -12393.347} C_VEL
LIN {X 0,Y 375.977,Z 492.776,A -85,B 0,C 180,E1 -12396.887,E2 -12396.887} C_VEL
LIN {X 0,Y 375.991,Z 492.762,A -85,B 0,C 180,E1 -12400.339,E2 -12400.339} C_VEL
LIN {X 0,Y 376.021,Z 492.768,A -85,B 0,C 180,E1 -12403.718,E2 -12403.718} C_VEL
LIN {X 0,Y 376.096,Z 492.738,A -85,B 0,C 180,E1 -12407.041,E2 -12407.041} C_VEL
LIN {X 0,Y 376.111,Z 492.758,A -85,B 0,C 180,E1 -12410.318,E2 -12410.318} C_VEL
LIN {X 0,Y 376.235,Z 492.721,A -85,B 0,C 180,E1 -12413.564,E2 -12413.564} C_VEL
LIN {X 0,Y 376.346,Z 492.729,A -85,B 0,C 180,E1 -12417.859,E2 -12417.859} C_VEL
LIN {X 0,Y 376.48,Z 492.702,A -85,B 0,C 180,E1 -12419.999,E2 -12419.999} C_VEL
LIN {X 0,Y 376.182,Z 492.73,A -85,B 0,C 180,E1 -12423.212,E2 -12423.212} C_VEL
LIN {X 0,Y 376.217,Z 492.741,A -85,B 0,C 180,E1 -12426.63,E2 -12426.63} C_VEL
LIN {X 0,Y 376.111,Z 492.737,A -85,B 0,C 180,E1 -12429.681,E2 -12429.681} C_VEL
LIN {X 0,Y 376.081,Z 492.766,A -85,B 0,C 180,E1 -12433.657,E2 -12433.657} C_VEL
LIN {X 0,Y 376.035,Z 492.75,A -85,B 0,C 180,E1 -12437.607,E2 -12437.607} C_VEL
LIN {X 0,Y 375.97,Z 492.775,A -85,B 0,C 180,E1 -12440.832,E2 -12440.832} C_VEL
LIN {X 0,Y 375.985,Z 492.756,A -85,B 0,C 180,E1 -12444.281,E2 -12444.281} C_VEL
LIN {X 0,Y 376.011,Z 492.769,A -85,B 0,C 180,E1 -12446.652,E2 -12446.652} C_VEL
LIN {X 0,Y 375.968,Z 492.774,A -85,B 0,C 180,E1 -12449.079,E2 -12449.079} C_VEL
LIN {X 0,Y 375.948,Z 492.778,A -85,B 0,C 180,E1 -12452.828,E2 -12452.828} C_VEL
LIN {X 0,Y 375.95,Z 492.771,A -85,B 0,C 180,E1 -12455.416,E2 -12455.416} C_VEL
LIN {X 0,Y 375.968,Z 492.778,A -85,B 0,C 180,E1 -12458.271,E2 -12458.271} C_VEL
LIN {X 0,Y 375.981,Z 492.768,A -85,B 0,C 180,E1 -12461.61,E2 -12461.61} C_VEL
LIN {X 0,Y 376.008,Z 492.751,A -85,B 0,C 180,E1 -12465.255,E2 -12465.255} C_VEL
LIN {X 0,Y 375.994,Z 492.767,A -85,B 0,C 180,E1 -12469.141,E2 -12469.141} C_VEL
LIN {X 0,Y 375.962,Z 492.764,A -85,B 0,C 180,E1 -12471.912,E2 -12471.912} C_VEL
LIN {X 0,Y 375.974,Z 492.774,A -85,B 0,C 180,E1 -12475.333,E2 -12475.333} C_VEL
LIN {X 0,Y 375.954,Z 492.781,A -85,B 0,C 180,E1 -12478.439,E2 -12478.439} C_VEL
LIN {X 0,Y 375.997,Z 492.776,A -85,B 0,C 180,E1 -12482.142,E2 -12482.142} C_VEL
LIN {X 0,Y 376.001,Z 492.776,A -85,B 0,C 180,E1 -12484.539,E2 -12484.539} C_VEL
LIN {X 0,Y 375.958,Z 492.781,A -85,B 0,C 180,E1 -12488.046,E2 -12488.046} C_VEL
LIN {X 0,Y 376.019,Z 492.773,A -85,B 0,C 180,E1 -12491.474,E2 -12491.474} C_VEL
LIN {X 0,Y 376.08,Z 493.029,A -85,B 0,C 180,E1 -12493.687,E2 -12493.687} C_VEL
LIN {X 0,Y 376.364,Z 494.161,A -85,B 0,C 180,E1 -12494.117,E2 -12494.117} C_VEL
LIN {X 0,Y 377.63,Z 496.441,A -85,B 0,C 180,E1 -12494.76,E2 -12494.76} C_VEL
LIN {X 0,Y 379.922,Z 498.234,A -85,B 0,C 180,E1 -12495.812,E2 -12495.812} C_VEL
LIN {X 0,Y 381.559,Z 499.252,A -85,B 0,C 180,E1 -12496.608,E2 -12496.608} C_VEL
LIN {X 0,Y 383.176,Z 502.133,A -85,B 0,C 180,E1 -12497.555,E2 -12497.555} C_VEL
LIN {X 0,Y 385.463,Z 504.119,A -85,B 0,C 180,E1 -12498.878,E2 -12498.878} C_VEL
LIN {X 0,Y 387.772,Z 505.431,A -85,B 0,C 180,E1 -12500.349,E2 -12500.349} C_VEL
LIN {X 0,Y 389.162,Z 507.674,A -85,B 0,C 180,E1 -12501.473,E2 -12501.473} C_VEL
LIN {X 0,Y 390.726,Z 509.469,A -85,B 0,C 180,E1 -12502.897,E2 -12502.897} C_VEL
LIN {X 0,Y 392.533,Z 510.682,A -85,B 0,C 180,E1 -12504.864,E2 -12504.864} C_VEL
LIN {X 0,Y 393.858,Z 511.178,A -85,B 0,C 180,E1 -12506.931,E2 -12506.931} C_VEL
LIN {X 0,Y 394.494,Z 511.664,A -85,B 0,C 180,E1 -12508.979,E2 -12508.979} C_VEL
LIN {X 0,Y 394.494,Z 511.667,A -85,B 0,C 180,E1 -12511.021,E2 -12511.021} C_VEL
LIN {X 0,Y 393.858,Z 511.175,A -85,B 0,C 180,E1 -12513.069,E2 -12513.069} C_VEL
LIN {X 0,Y 392.536,Z 510.666,A -85,B 0,C 180,E1 -12515.136,E2 -12515.136} C_VEL
LIN {X 0,Y 390.6,Z 509.302,A -85,B 0,C 180,E1 -12517.235,E2 -12517.235} C_VEL
LIN {X 0,Y 388.843,Z 507.315,A -85,B 0,C 180,E1 -12518.773,E2 -12518.773} C_VEL
LIN {X 0,Y 387.374,Z 505.064,A -85,B 0,C 180,E1 -12519.925,E2 -12519.925} C_VEL
LIN {X 0,Y 384.403,Z 503.362,A -85,B 0,C 180,E1 -12521.735,E2 -12521.735} C_VEL
LIN {X 0,Y 382.596,Z 501.268,A -85,B 0,C 180,E1 -12522.778,E2 -12522.778} C_VEL
LIN {X 0,Y 381.274,Z 498.917,A -85,B 0,C 180,E1 -12523.539,E2 -12523.539} C_VEL
LIN {X 0,Y 378.402,Z 497.208,A -85,B 0,C 180,E1 -12524.886,E2 -12524.886} C_VEL
LIN {X 0,Y 376.824,Z 495.266,A -85,B 0,C 180,E1 -12525.62,E2 -12525.62} C_VEL
LIN {X 0,Y 376.139,Z 493.326,A -85,B 0,C 180,E1 -12526.136,E2 -12526.136} C_VEL
LIN {X 0,Y 376.063,Z 492.784,A -85,B 0,C 180,E1 -12526.838,E2 -12526.838} C_VEL
LIN {X 0,Y 375.993,Z 492.777,A -85,B 0,C 180,E1 -12529.66,E2 -12529.66} C_VEL
LIN {X 0,Y 375.991,Z 492.777,A -85,B 0,C 180,E1 -12533.667,E2 -12533.667} C_VEL
LIN {X 0,Y 376.014,Z 492.774,A -85,B 0,C 180,E1 -12536.652,E2 -12536.652} C_VEL
LIN {X 0,Y 375.971,Z 492.778,A -85,B 0,C 180,E1 -12539.078,E2 -12539.078} C_VEL
LIN {X 0,Y 375.945,Z 492.782,A -85,B 0,C 180,E1 -12542.828,E2 -12542.828} C_VEL
LIN {X 0,Y 375.952,Z 492.766,A -85,B 0,C 180,E1 -12545.415,E2 -12545.415} C_VEL
LIN {X 0,Y 375.972,Z 492.765,A -85,B 0,C 180,E1 -12548.271,E2 -12548.271} C_VEL
LIN {X 0,Y 375.99,Z 492.777,A -85,B 0,C 180,E1 -12550.043,E2 -12550.043} C_VEL
LIN {X 0,Y 375.297,Z 492.854,A -85,B 0,C 180,E1 -12550.936,E2 -12550.936} C_VEL
LIN {X 0,Y 372.421,Z 493.186,A -85,B 0,C 180,E1 -12552.39,E2 -12552.39} C_VEL
LIN {X 0,Y 370.027,Z 493.48,A -85,B 0,C 180,E1 -12553.565,E2 -12553.565} C_VEL
LIN {X 0,Y 369.04,Z 493.612,A -85,B 0,C 180,E1 -12554.474,E2 -12554.474} C_VEL
LIN {X 0,Y 368.981,Z 493.626,A -85,B 0,C 180,E1 -12554.782,E2 -12554.782} C_VEL
LIN {X 0,Y 368.937,Z 493.648,A -85,B 0,C 180,E1 -12558.186,E2 -12558.186} C_VEL
LIN {X 0,Y 368.903,Z 493.657,A -85,B 0,C 180,E1 -12561.359,E2 -12561.359} C_VEL
LIN {X 0,Y 368.929,Z 493.649,A -85,B 0,C 180,E1 -12565.146,E2 -12565.146} C_VEL
LIN {X 0,Y 368.921,Z 493.638,A -85,B 0,C 180,E1 -12569.046,E2 -12569.046} C_VEL
LIN {X 0,Y 368.978,Z 493.644,A -85,B 0,C 180,E1 -12571.565,E2 -12571.565} C_VEL
LIN {X 0,Y 368.949,Z 493.634,A -85,B 0,C 180,E1 -12575.225,E2 -12575.225} C_VEL
LIN {X 0,Y 368.929,Z 493.653,A -85,B 0,C 180,E1 -12578.973,E2 -12578.973} C_VEL
LIN {X 0,Y 368.982,Z 493.628,A -85,B 0,C 180,E1 -12582.257,E2 -12582.257} C_VEL
LIN {X 0,Y 369.028,Z 493.643,A -85,B 0,C 180,E1 -12586.228,E2 -12586.228} C_VEL
LIN {X 0,Y 369.059,Z 493.615,A -85,B 0,C 180,E1 -12590.132,E2 -12590.132} C_VEL
LIN {X 0,Y 369.198,Z 493.617,A -85,B 0,C 180,E1 -12593.442,E2 -12593.442} C_VEL
LIN {X 0,Y 369.311,Z 493.58,A -85,B 0,C 180,E1 -12597.819,E2 -12597.819} C_VEL
LIN {X 0,Y 369.45,Z 493.578,A -85,B 0,C 180,E1 -12600.001,E2 -12600.001} C_VEL
LIN {X 0,Y 369.311,Z 493.606,A -85,B 0,C 180,E1 -12602.182,E2 -12602.182} C_VEL
LIN {X 0,Y 369.195,Z 493.599,A -85,B 0,C 180,E1 -12606.559,E2 -12606.559} C_VEL
LIN {X 0,Y 369.114,Z 493.632,A -85,B 0,C 180,E1 -12608.762,E2 -12608.762} C_VEL
LIN {X 0,Y 368.998,Z 493.633,A -85,B 0,C 180,E1 -12612.094,E2 -12612.094} C_VEL
LIN {X 0,Y 368.99,Z 493.64,A -85,B 0,C 180,E1 -12615.466,E2 -12615.466} C_VEL
LIN {X 0,Y 368.96,Z 493.641,A -85,B 0,C 180,E1 -12618.894,E2 -12618.894} C_VEL
LIN {X 0,Y 368.918,Z 493.646,A -85,B 0,C 180,E1 -12622.396,E2 -12622.396} C_VEL
LIN {X 0,Y 368.994,Z 493.639,A -85,B 0,C 180,E1 -12625.981,E2 -12625.981} C_VEL
LIN {X 0,Y 368.909,Z 493.654,A -85,B 0,C 180,E1 -12629.691,E2 -12629.691} C_VEL
LIN {X 0,Y 368.892,Z 493.645,A -85,B 0,C 180,E1 -12633.044,E2 -12633.044} C_VEL
LIN {X 0,Y 368.914,Z 493.657,A -85,B 0,C 180,E1 -12636.198,E2 -12636.198} C_VEL
LIN {X 0,Y 368.905,Z 493.654,A -85,B 0,C 180,E1 -12638.953,E2 -12638.953} C_VEL
LIN {X 0,Y 368.906,Z 493.65,A -85,B 0,C 180,E1 -12642.015,E2 -12642.015} C_VEL
LIN {X 0,Y 368.878,Z 493.652,A -85,B 0,C 180,E1 -12645.177,E2 -12645.177} C_VEL
LIN {X 0,Y 368.881,Z 493.651,A -85,B 0,C 180,E1 -12648.179,E2 -12648.179} C_VEL
LIN {X 0,Y 368.907,Z 493.621,A -85,B 0,C 180,E1 -12651.361,E2 -12651.361} C_VEL
LIN {X 0,Y 368.935,Z 493.608,A -85,B 0,C 180,E1 -12655.147,E2 -12655.147} C_VEL
LIN {X 0,Y 368.961,Z 493.857,A -85,B 0,C 180,E1 -12655.895,E2 -12655.895} C_VEL
LIN {X 0,Y 370.853,Z 502.314,A -85,B 0,C 180,E1 -12658.517,E2 -12658.517} C_VEL
LIN {X 0,Y 373.042,Z 513.149,A -85,B 0,C 180,E1 -12661.596,E2 -12661.596} C_VEL
LIN {X 0,Y 373.377,Z 517.039,A -85,B 0,C 180,E1 -12662.679,E2 -12662.679} C_VEL
LIN {X 0,Y 372.995,Z 520.963,A -85,B 0,C 180,E1 -12663.663,E2 -12663.663} C_VEL
LIN {X 0,Y 376.799,Z 537.609,A -85,B 0,C 180,E1 -12664.329,E2 -12664.329} C_VEL
LIN {X 0,Y 381.186,Z 560.065,A -85,B 0,C 180,E1 -12665.1,E2 -12665.1} C_VEL
LIN {X 0,Y 379.331,Z 653.813,A -85,B 0,C 180,E1 -12666.887,E2 -12666.887} C_VEL
LIN {X 0,Y 378.824,Z 665.576,A -85,B 0,C 180,E1 -12667.215,E2 -12667.215} C_VEL
LIN {X 0,Y 378.076,Z 677.03,A -85,B 0,C 180,E1 -12667.673,E2 -12667.673} C_VEL
LIN {X 0,Y 377.205,Z 688.184,A -85,B 0,C 180,E1 -12668.266,E2 -12668.266} C_VEL
LIN {X 0,Y 376.325,Z 698.157,A -85,B 0,C 180,E1 -12668.931,E2 -12668.931} C_VEL
LIN {X 0,Y 375.346,Z 708.054,A -85,B 0,C 180,E1 -12669.731,E2 -12669.731} C_VEL
LIN {X 0,Y 374.232,Z 717.805,A -85,B 0,C 180,E1 -12670.671,E2 -12670.671} C_VEL
LIN {X 0,Y 373.004,Z 727.223,A -85,B 0,C 180,E1 -12671.746,E2 -12671.746} C_VEL
LIN {X 0,Y 371.9,Z 736.248,A -85,B 0,C 180,E1 -12672.968,E2 -12672.968} C_VEL
LIN {X 0,Y 370.978,Z 743.223,A -85,B 0,C 180,E1 -12674.057,E2 -12674.057} C_VEL
LIN {X 0,Y 370.08,Z 750.75,A -85,B 0,C 180,E1 -12675.427,E2 -12675.427} C_VEL
LIN {X 0,Y 369.237,Z 758.366,A -85,B 0,C 180,E1 -12677.077,E2 -12677.077} C_VEL
LIN {X 0,Y 368.622,Z 763.769,A -85,B 0,C 180,E1 -12678.452,E2 -12678.452} C_VEL
LIN {X 0,Y 368.079,Z 769.202,A -85,B 0,C 180,E1 -12680.105,E2 -12680.105} C_VEL
LIN {X 0,Y 367.736,Z 773.647,A -85,B 0,C 180,E1 -12681.759,E2 -12681.759} C_VEL
LIN {X 0,Y 367.557,Z 777.192,A -85,B 0,C 180,E1 -12683.412,E2 -12683.412} C_VEL
LIN {X 0,Y 367.447,Z 779.131,A -85,B 0,C 180,E1 -12684.512,E2 -12684.512} C_VEL
LIN {X 0,Y 367.372,Z 781.814,A -85,B 0,C 180,E1 -12686.71,E2 -12686.71} C_VEL
LIN {X 0,Y 367.415,Z 783.104,A -85,B 0,C 180,E1 -12688.904,E2 -12688.904} C_VEL
LIN {X 0,Y 367.456,Z 783.357,A -85,B 0,C 180,E1 -12690,E2 -12690} C_VEL
LIN {X 0,Y 367.357,Z 782.63,A -85,B 0,C 180,E1 -12692.193,E2 -12692.193} C_VEL
LIN {X 0,Y 367.372,Z 781.814,A -85,B 0,C 180,E1 -12693.29,E2 -12693.29} C_VEL
LIN {X 0,Y 367.447,Z 779.131,A -85,B 0,C 180,E1 -12695.488,E2 -12695.488} C_VEL
LIN {X 0,Y 367.597,Z 776.176,A -85,B 0,C 180,E1 -12697.139,E2 -12697.139} C_VEL
LIN {X 0,Y 367.819,Z 772.349,A -85,B 0,C 180,E1 -12698.792,E2 -12698.792} C_VEL
LIN {X 0,Y 368.211,Z 767.585,A -85,B 0,C 180,E1 -12700.447,E2 -12700.447} C_VEL
LIN {X 0,Y 369.007,Z 760.642,A -85,B 0,C 180,E1 -12702.372,E2 -12702.372} C_VEL
LIN {X 0,Y 369.631,Z 755.036,A -85,B 0,C 180,E1 -12703.692,E2 -12703.692} C_VEL
LIN {X 0,Y 370.434,Z 747.911,A -85,B 0,C 180,E1 -12705.121,E2 -12705.121} C_VEL
LIN {X 0,Y 371.421,Z 739.885,A -85,B 0,C 180,E1 -12706.488,E2 -12706.488} C_VEL
LIN {X 0,Y 372.593,Z 730.403,A -85,B 0,C 180,E1 -12707.849,E2 -12707.849} C_VEL
LIN {X 0,Y 373.74,Z 721.525,A -85,B 0,C 180,E1 -12708.927,E2 -12708.927} C_VEL
LIN {X 0,Y 374.977,Z 711.404,A -85,B 0,C 180,E1 -12709.963,E2 -12709.963} C_VEL
LIN {X 0,Y 375.975,Z 701.337,A -85,B 0,C 180,E1 -12710.83,E2 -12710.83} C_VEL
LIN {X 0,Y 376.98,Z 690.761,A -85,B 0,C 180,E1 -12711.575,E2 -12711.575} C_VEL
LIN {X 0,Y 377.846,Z 679.749,A -85,B 0,C 180,E1 -12712.198,E2 -12712.198} C_VEL
LIN {X 0,Y 378.639,Z 669.225,A -85,B 0,C 180,E1 -12712.652,E2 -12712.652} C_VEL
LIN {X 0,Y 379.198,Z 657.809,A -85,B 0,C 180,E1 -12713.013,E2 -12713.013} C_VEL
LIN {X 0,Y 379.982,Z 627.699,A -85,B 0,C 180,E1 -12713.612,E2 -12713.612} C_VEL
LIN {X 0,Y 381.109,Z 559.496,A -85,B 0,C 180,E1 -12714.917,E2 -12714.917} C_VEL
LIN {X 0,Y 375.789,Z 533.154,A -85,B 0,C 180,E1 -12715.837,E2 -12715.837} C_VEL
LIN {X 0,Y 373.016,Z 520.976,A -85,B 0,C 180,E1 -12716.333,E2 -12716.333} C_VEL
LIN {X 0,Y 373.386,Z 515.305,A -85,B 0,C 180,E1 -12717.791,E2 -12717.791} C_VEL
LIN {X 0,Y 371.436,Z 505.079,A -85,B 0,C 180,E1 -12720.721,E2 -12720.721} C_VEL
LIN {X 0,Y 368.958,Z 493.836,A -85,B 0,C 180,E1 -12724.106,E2 -12724.106} C_VEL
LIN {X 0,Y 368.9,Z 493.593,A -85,B 0,C 180,E1 -12726.855,E2 -12726.855} C_VEL
LIN {X 0,Y 368.91,Z 493.657,A -85,B 0,C 180,E1 -12730.369,E2 -12730.369} C_VEL
LIN {X 0,Y 368.88,Z 493.637,A -85,B 0,C 180,E1 -12733.615,E2 -12733.615} C_VEL
LIN {X 0,Y 368.901,Z 493.659,A -85,B 0,C 180,E1 -12736.698,E2 -12736.698} C_VEL
LIN {X 0,Y 368.95,Z 493.653,A -85,B 0,C 180,E1 -12739.635,E2 -12739.635} C_VEL
LIN {X 0,Y 368.899,Z 493.653,A -85,B 0,C 180,E1 -12743.143,E2 -12743.143} C_VEL
LIN {X 0,Y 368.892,Z 493.647,A -85,B 0,C 180,E1 -12746.461,E2 -12746.461} C_VEL
LIN {X 0,Y 368.924,Z 493.653,A -85,B 0,C 180,E1 -12749.046,E2 -12749.046} C_VEL
LIN {X 0,Y 368.957,Z 493.633,A -85,B 0,C 180,E1 -12752.796,E2 -12752.796} C_VEL
LIN {X 0,Y 368.931,Z 493.652,A -85,B 0,C 180,E1 -12756.115,E2 -12756.115} C_VEL
LIN {X 0,Y 368.923,Z 493.638,A -85,B 0,C 180,E1 -12759.946,E2 -12759.946} C_VEL
LIN {X 0,Y 368.969,Z 493.65,A -85,B 0,C 180,E1 -12763.398,E2 -12763.398} C_VEL
LIN {X 0,Y 369.05,Z 493.614,A -85,B 0,C 180,E1 -12766.789,E2 -12766.789} C_VEL
LIN {X 0,Y 369.06,Z 493.637,A -85,B 0,C 180,E1 -12770.131,E2 -12770.131} C_VEL
LIN {X 0,Y 369.157,Z 493.616,A -85,B 0,C 180,E1 -12772.341,E2 -12772.341} C_VEL
LIN {X 0,Y 369.136,Z 493.602,A -85,B 0,C 180,E1 -12774.537,E2 -12774.537} C_VEL
LIN {X 0,Y 369.311,Z 493.606,A -85,B 0,C 180,E1 -12777.818,E2 -12777.818} C_VEL
LIN {X 0,Y 369.45,Z 493.578,A -85,B 0,C 180,E1 -12779.999,E2 -12779.999} C_VEL
LIN {X 0,Y 369.311,Z 493.58,A -85,B 0,C 180,E1 -12782.181,E2 -12782.181} C_VEL
LIN {X 0,Y 369.187,Z 493.617,A -85,B 0,C 180,E1 -12786.615,E2 -12786.615} C_VEL
LIN {X 0,Y 369.059,Z 493.615,A -85,B 0,C 180,E1 -12789.868,E2 -12789.868} C_VEL
LIN {X 0,Y 369.028,Z 493.643,A -85,B 0,C 180,E1 -12793.772,E2 -12793.772} C_VEL
LIN {X 0,Y 368.993,Z 493.627,A -85,B 0,C 180,E1 -12797.768,E2 -12797.768} C_VEL
LIN {X 0,Y 368.922,Z 493.655,A -85,B 0,C 180,E1 -12801.219,E2 -12801.219} C_VEL
LIN {X 0,Y 368.949,Z 493.634,A -85,B 0,C 180,E1 -12804.775,E2 -12804.775} C_VEL
LIN {X 0,Y 368.978,Z 493.644,A -85,B 0,C 180,E1 -12808.435,E2 -12808.435} C_VEL
LIN {X 0,Y 368.901,Z 493.657,A -85,B 0,C 180,E1 -12812.237,E2 -12812.237} C_VEL
LIN {X 0,Y 368.921,Z 493.65,A -85,B 0,C 180,E1 -12815.002,E2 -12815.002} C_VEL
LIN {X 0,Y 368.903,Z 493.657,A -85,B 0,C 180,E1 -12818.641,E2 -12818.641} C_VEL
LIN {X 0,Y 368.943,Z 493.65,A -85,B 0,C 180,E1 -12822.022,E2 -12822.022} C_VEL
LIN {X 0,Y 368.983,Z 493.626,A -85,B 0,C 180,E1 -12825.193,E2 -12825.193} C_VEL
LIN {X 0,Y 368.934,Z 493.625,A -85,B 0,C 180,E1 -12828.186,E2 -12828.186} C_VEL
LIN {X 0,Y 368.908,Z 493.651,A -85,B 0,C 180,E1 -12831.359,E2 -12831.359} C_VEL
LIN {X 0,Y 368.931,Z 493.651,A -85,B 0,C 180,E1 -12835.147,E2 -12835.147} C_VEL
LIN {X 0,Y 368.923,Z 493.656,A -85,B 0,C 180,E1 -12839.047,E2 -12839.047} C_VEL
LIN {X 0,Y 368.981,Z 493.65,A -85,B 0,C 180,E1 -12841.565,E2 -12841.565} C_VEL
LIN {X 0,Y 368.953,Z 493.653,A -85,B 0,C 180,E1 -12845.225,E2 -12845.225} C_VEL
LIN {X 0,Y 368.933,Z 493.656,A -85,B 0,C 180,E1 -12848.974,E2 -12848.974} C_VEL
LIN {X 0,Y 369.015,Z 493.915,A -85,B 0,C 180,E1 -12851.239,E2 -12851.239} C_VEL
LIN {X 0,Y 369.266,Z 494.925,A -85,B 0,C 180,E1 -12851.608,E2 -12851.608} C_VEL
LIN {X 0,Y 370.704,Z 497.466,A -85,B 0,C 180,E1 -12852.225,E2 -12852.225} C_VEL
LIN {X 0,Y 373.238,Z 499.31,A -85,B 0,C 180,E1 -12853.214,E2 -12853.214} C_VEL
LIN {X 0,Y 374.251,Z 500.169,A -85,B 0,C 180,E1 -12853.64,E2 -12853.64} C_VEL
LIN {X 0,Y 375.892,Z 502.925,A -85,B 0,C 180,E1 -12854.409,E2 -12854.409} C_VEL
LIN {X 0,Y 378.234,Z 504.929,A -85,B 0,C 180,E1 -12855.472,E2 -12855.472} C_VEL
LIN {X 0,Y 380,Z 505.963,A -85,B 0,C 180,E1 -12856.298,E2 -12856.298} C_VEL
LIN {X 0,Y 381.802,Z 508.909,A -85,B 0,C 180,E1 -12857.312,E2 -12857.312} C_VEL
LIN {X 0,Y 384.118,Z 510.907,A -85,B 0,C 180,E1 -12858.614,E2 -12858.614} C_VEL
LIN {X 0,Y 386.626,Z 512.443,A -85,B 0,C 180,E1 -12860.188,E2 -12860.188} C_VEL
LIN {X 0,Y 388.232,Z 514.832,A -85,B 0,C 180,E1 -12861.452,E2 -12861.452} C_VEL
LIN {X 0,Y 389.967,Z 516.641,A -85,B 0,C 180,E1 -12863.013,E2 -12863.013} C_VEL
LIN {X 0,Y 391.853,Z 517.829,A -85,B 0,C 180,E1 -12865.102,E2 -12865.102} C_VEL
LIN {X 0,Y 393.179,Z 518.343,A -85,B 0,C 180,E1 -12867.346,E2 -12867.346} C_VEL
LIN {X 0,Y 393.631,Z 518.69,A -85,B 0,C 180,E1 -12868.977,E2 -12868.977} C_VEL
LIN {X 0,Y 393.627,Z 518.701,A -85,B 0,C 180,E1 -12871.035,E2 -12871.035} C_VEL
LIN {X 0,Y 392.988,Z 518.211,A -85,B 0,C 180,E1 -12873.075,E2 -12873.075} C_VEL
LIN {X 0,Y 391.655,Z 517.718,A -85,B 0,C 180,E1 -12875.147,E2 -12875.147} C_VEL
LIN {X 0,Y 389.675,Z 516.368,A -85,B 0,C 180,E1 -12877.278,E2 -12877.278} C_VEL
LIN {X 0,Y 387.914,Z 514.469,A -85,B 0,C 180,E1 -12878.794,E2 -12878.794} C_VEL
LIN {X 0,Y 386.245,Z 511.986,A -85,B 0,C 180,E1 -12880.086,E2 -12880.086} C_VEL
LIN {X 0,Y 383.317,Z 510.38,A -85,B 0,C 180,E1 -12881.836,E2 -12881.836} C_VEL
LIN {X 0,Y 381.121,Z 507.96,A -85,B 0,C 180,E1 -12883.082,E2 -12883.082} C_VEL
LIN {X 0,Y 379.869,Z 505.718,A -85,B 0,C 180,E1 -12883.777,E2 -12883.777} C_VEL
LIN {X 0,Y 376.921,Z 503.96,A -85,B 0,C 180,E1 -12885.132,E2 -12885.132} C_VEL
LIN {X 0,Y 374.913,Z 501.492,A -85,B 0,C 180,E1 -12886.051,E2 -12886.051} C_VEL
LIN {X 0,Y 373.873,Z 499.63,A -85,B 0,C 180,E1 -12886.529,E2 -12886.529} C_VEL
LIN {X 0,Y 370.921,Z 497.696,A -85,B 0,C 180,E1 -12887.686,E2 -12887.686} C_VEL
LIN {X 0,Y 369.402,Z 495.352,A -85,B 0,C 180,E1 -12888.317,E2 -12888.317} C_VEL
LIN {X 0,Y 369.047,Z 494.148,A -85,B 0,C 180,E1 -12888.63,E2 -12888.63} C_VEL
LIN {X 0,Y 368.945,Z 493.681,A -85,B 0,C 180,E1 -12889.183,E2 -12889.183} C_VEL
LIN {X 0,Y 368.927,Z 493.657,A -85,B 0,C 180,E1 -12892.395,E2 -12892.395} C_VEL
LIN {X 0,Y 368.995,Z 493.648,A -85,B 0,C 180,E1 -12895.98,E2 -12895.98} C_VEL
LIN {X 0,Y 368.962,Z 493.652,A -85,B 0,C 180,E1 -12898.813,E2 -12898.813} C_VEL
LIN {X 0,Y 368.894,Z 493.662,A -85,B 0,C 180,E1 -12902.238,E2 -12902.238} C_VEL
LIN {X 0,Y 368.923,Z 493.649,A -85,B 0,C 180,E1 -12905.001,E2 -12905.001} C_VEL
LIN {X 0,Y 368.907,Z 493.651,A -85,B 0,C 180,E1 -12908.641,E2 -12908.641} C_VEL
LIN {X 0,Y 368.935,Z 493.621,A -85,B 0,C 180,E1 -12912.02,E2 -12912.02} C_VEL
LIN {X 0,Y 368.981,Z 493.626,A -85,B 0,C 180,E1 -12914.782,E2 -12914.782} C_VEL
LIN {X 0,Y 368.365,Z 493.719,A -85,B 0,C 180,E1 -12915.692,E2 -12915.692} C_VEL
LIN {X 0,Y 365.508,Z 494.08,A -85,B 0,C 180,E1 -12917.172,E2 -12917.172} C_VEL
LIN {X 0,Y 363.044,Z 494.379,A -85,B 0,C 180,E1 -12918.369,E2 -12918.369} C_VEL
LIN {X 0,Y 361.97,Z 494.509,A -85,B 0,C 180,E1 -12919.295,E2 -12919.295} C_VEL
LIN {X 0,Y 361.877,Z 494.521,A -85,B 0,C 180,E1 -12919.609,E2 -12919.609} C_VEL
LIN {X 0,Y 361.861,Z 494.527,A -85,B 0,C 180,E1 -12922.982,E2 -12922.982} C_VEL
LIN {X 0,Y 361.854,Z 494.536,A -85,B 0,C 180,E1 -12926.63,E2 -12926.63} C_VEL
LIN {X 0,Y 361.869,Z 494.516,A -85,B 0,C 180,E1 -12929.672,E2 -12929.672} C_VEL
LIN {X 0,Y 361.946,Z 494.521,A -85,B 0,C 180,E1 -12933.475,E2 -12933.475} C_VEL
LIN {X 0,Y 361.883,Z 494.525,A -85,B 0,C 180,E1 -12937.145,E2 -12937.145} C_VEL
LIN {X 0,Y 361.903,Z 494.52,A -85,B 0,C 180,E1 -12940.724,E2 -12940.724} C_VEL
LIN {X 0,Y 361.924,Z 494.507,A -85,B 0,C 180,E1 -12943.066,E2 -12943.066} C_VEL
LIN {X 0,Y 361.99,Z 494.52,A -85,B 0,C 180,E1 -12946.528,E2 -12946.528} C_VEL
LIN {X 0,Y 362.023,Z 494.491,A -85,B 0,C 180,E1 -12949.938,E2 -12949.938} C_VEL
LIN {X 0,Y 362.159,Z 494.494,A -85,B 0,C 180,E1 -12953.314,E2 -12953.314} C_VEL
LIN {X 0,Y 362.275,Z 494.456,A -85,B 0,C 180,E1 -12957.777,E2 -12957.777} C_VEL
LIN {X 0,Y 362.419,Z 494.453,A -85,B 0,C 180,E1 -12960.001,E2 -12960.001} C_VEL
LIN {X 0,Y 362.275,Z 494.482,A -85,B 0,C 180,E1 -12962.224,E2 -12962.224} C_VEL
LIN {X 0,Y 362.157,Z 494.476,A -85,B 0,C 180,E1 -12966.687,E2 -12966.687} C_VEL
LIN {X 0,Y 362.024,Z 494.514,A -85,B 0,C 180,E1 -12970.063,E2 -12970.063} C_VEL
LIN {X 0,Y 361.991,Z 494.493,A -85,B 0,C 180,E1 -12973.899,E2 -12973.899} C_VEL
LIN {X 0,Y 361.961,Z 494.521,A -85,B 0,C 180,E1 -12977.939,E2 -12977.939} C_VEL
LIN {X 0,Y 361.856,Z 494.522,A -85,B 0,C 180,E1 -12981.656,E2 -12981.656} C_VEL
LIN {X 0,Y 361.921,Z 494.521,A -85,B 0,C 180,E1 -12985.291,E2 -12985.291} C_VEL
LIN {X 0,Y 361.903,Z 494.514,A -85,B 0,C 180,E1 -12987.78,E2 -12987.78} C_VEL
LIN {X 0,Y 361.833,Z 494.532,A -85,B 0,C 180,E1 -12991.63,E2 -12991.63} C_VEL
LIN {X 0,Y 361.87,Z 494.533,A -85,B 0,C 180,E1 -12995.346,E2 -12995.346} C_VEL
LIN {X 0,Y 361.871,Z 494.531,A -85,B 0,C 180,E1 -12999.029,E2 -12999.029} C_VEL
LIN {X 0,Y 361.853,Z 494.53,A -85,B 0,C 180,E1 -13002.436,E2 -13002.436} C_VEL
LIN {X 0,Y 361.816,Z 494.521,A -85,B 0,C 180,E1 -13005.947,E2 -13005.947} C_VEL
LIN {X 0,Y 361.835,Z 494.54,A -85,B 0,C 180,E1 -13009.245,E2 -13009.245} C_VEL
LIN {X 0,Y 361.862,Z 494.47,A -85,B 0,C 180,E1 -13012.778,E2 -13012.778} C_VEL
LIN {X 0,Y 361.906,Z 494.611,A -85,B 0,C 180,E1 -13015.389,E2 -13015.389} C_VEL
LIN {X 0,Y 363.317,Z 501.02,A -85,B 0,C 180,E1 -13017.489,E2 -13017.489} C_VEL
LIN {X 0,Y 365.585,Z 511.791,A -85,B 0,C 180,E1 -13020.646,E2 -13020.646} C_VEL
LIN {X 0,Y 366.477,Z 517.348,A -85,B 0,C 180,E1 -13022.269,E2 -13022.269} C_VEL
LIN {X 0,Y 366.216,Z 520.809,A -85,B 0,C 180,E1 -13023.143,E2 -13023.143} C_VEL
LIN {X 0,Y 370.782,Z 540.815,A -85,B 0,C 180,E1 -13023.953,E2 -13023.953} C_VEL
LIN {X 0,Y 374.772,Z 561.793,A -85,B 0,C 180,E1 -13024.684,E2 -13024.684} C_VEL
LIN {X 0,Y 372.758,Z 656.253,A -85,B 0,C 180,E1 -13026.529,E2 -13026.529} C_VEL
LIN {X 0,Y 372.191,Z 667.202,A -85,B 0,C 180,E1 -13026.859,E2 -13026.859} C_VEL
LIN {X 0,Y 371.417,Z 678.192,A -85,B 0,C 180,E1 -13027.323,E2 -13027.323} C_VEL
LIN {X 0,Y 370.582,Z 687.985,A -85,B 0,C 180,E1 -13027.857,E2 -13027.857} C_VEL
LIN {X 0,Y 369.699,Z 697.959,A -85,B 0,C 180,E1 -13028.535,E2 -13028.535} C_VEL
LIN {X 0,Y 368.697,Z 707.491,A -85,B 0,C 180,E1 -13029.313,E2 -13029.313} C_VEL
LIN {X 0,Y 367.509,Z 717.606,A -85,B 0,C 180,E1 -13030.303,E2 -13030.303} C_VEL
LIN {X 0,Y 366.244,Z 727.025,A -85,B 0,C 180,E1 -13031.397,E2 -13031.397} C_VEL
LIN {X 0,Y 365.081,Z 736.048,A -85,B 0,C 180,E1 -13032.64,E2 -13032.64} C_VEL
LIN {X 0,Y 364.107,Z 743.024,A -85,B 0,C 180,E1 -13033.747,E2 -13033.747} C_VEL
LIN {X 0,Y 363.161,Z 750.55,A -85,B 0,C 180,E1 -13035.143,E2 -13035.143} C_VEL
LIN {X 0,Y 362.401,Z 757.028,A -85,B 0,C 180,E1 -13036.543,E2 -13036.543} C_VEL
LIN {X 0,Y 361.631,Z 763.57,A -85,B 0,C 180,E1 -13038.226,E2 -13038.226} C_VEL
LIN {X 0,Y 361.031,Z 769.002,A -85,B 0,C 180,E1 -13039.91,E2 -13039.91} C_VEL
LIN {X 0,Y 360.662,Z 773.448,A -85,B 0,C 180,E1 -13041.596,E2 -13041.596} C_VEL
LIN {X 0,Y 360.487,Z 776.994,A -85,B 0,C 180,E1 -13043.283,E2 -13043.283} C_VEL
LIN {X 0,Y 360.355,Z 778.933,A -85,B 0,C 180,E1 -13044.404,E2 -13044.404} C_VEL
LIN {X 0,Y 360.291,Z 781.616,A -85,B 0,C 180,E1 -13046.645,E2 -13046.645} C_VEL
LIN {X 0,Y 360.315,Z 782.906,A -85,B 0,C 180,E1 -13048.882,E2 -13048.882} C_VEL
LIN {X 0,Y 360.359,Z 783.159,A -85,B 0,C 180,E1 -13050,E2 -13050} C_VEL
LIN {X 0,Y 360.262,Z 782.432,A -85,B 0,C 180,E1 -13052.236,E2 -13052.236} C_VEL
LIN {X 0,Y 360.291,Z 781.616,A -85,B 0,C 180,E1 -13053.355,E2 -13053.355} C_VEL
LIN {X 0,Y 360.356,Z 778.933,A -85,B 0,C 180,E1 -13055.596,E2 -13055.596} C_VEL
LIN {X 0,Y 360.511,Z 775.977,A -85,B 0,C 180,E1 -13057.28,E2 -13057.28} C_VEL
LIN {X 0,Y 360.774,Z 772.15,A -85,B 0,C 180,E1 -13058.965,E2 -13058.965} C_VEL
LIN {X 0,Y 361.187,Z 767.386,A -85,B 0,C 180,E1 -13060.652,E2 -13060.652} C_VEL
LIN {X 0,Y 362.037,Z 760.443,A -85,B 0,C 180,E1 -13062.614,E2 -13062.614} C_VEL
LIN {X 0,Y 362.772,Z 753.693,A -85,B 0,C 180,E1 -13064.2,E2 -13064.2} C_VEL
LIN {X 0,Y 363.699,Z 746.149,A -85,B 0,C 180,E1 -13065.695,E2 -13065.695} C_VEL
LIN {X 0,Y 364.8,Z 737.866,A -85,B 0,C 180,E1 -13067.085,E2 -13067.085} C_VEL
LIN {X 0,Y 365.961,Z 729.144,A -85,B 0,C 180,E1 -13068.328,E2 -13068.328} C_VEL
LIN {X 0,Y 367.197,Z 720.087,A -85,B 0,C 180,E1 -13069.423,E2 -13069.423} C_VEL
LIN {X 0,Y 368.278,Z 711.407,A -85,B 0,C 180,E1 -13070.322,E2 -13070.322} C_VEL
LIN {X 0,Y 369.311,Z 701.466,A -85,B 0,C 180,E1 -13071.196,E2 -13071.196} C_VEL
LIN {X 0,Y 370.33,Z 691.207,A -85,B 0,C 180,E1 -13071.939,E2 -13071.939} C_VEL
LIN {X 0,Y 371.17,Z 680.911,A -85,B 0,C 180,E1 -13072.546,E2 -13072.546} C_VEL
LIN {X 0,Y 372.078,Z 669.026,A -85,B 0,C 180,E1 -13073.074,E2 -13073.074} C_VEL
LIN {X 0,Y 372.673,Z 657.611,A -85,B 0,C 180,E1 -13073.44,E2 -13073.44} C_VEL
LIN {X 0,Y 373.5,Z 627.501,A -85,B 0,C 180,E1 -13074.047,E2 -13074.047} C_VEL
LIN {X 0,Y 374.715,Z 560.838,A -85,B 0,C 180,E1 -13075.34,E2 -13075.34} C_VEL
LIN {X 0,Y 369.399,Z 534.369,A -85,B 0,C 180,E1 -13076.287,E2 -13076.287} C_VEL
LIN {X 0,Y 366.254,Z 520.902,A -85,B 0,C 180,E1 -13076.845,E2 -13076.845} C_VEL
LIN {X 0,Y 366.455,Z 518.514,A -85,B 0,C 180,E1 -13077.405,E2 -13077.405} C_VEL
LIN {X 0,Y 366.016,Z 514.048,A -85,B 0,C 180,E1 -13078.687,E2 -13078.687} C_VEL
LIN {X 0,Y 363.901,Z 503.483,A -85,B 0,C 180,E1 -13081.813,E2 -13081.813} C_VEL
LIN {X 0,Y 361.906,Z 494.599,A -85,B 0,C 180,E1 -13084.611,E2 -13084.611} C_VEL
LIN {X 0,Y 361.867,Z 494.49,A -85,B 0,C 180,E1 -13088.424,E2 -13088.424} C_VEL
LIN {X 0,Y 361.826,Z 494.535,A -85,B 0,C 180,E1 -13091.33,E2 -13091.33} C_VEL
LIN {X 0,Y 361.815,Z 494.524,A -85,B 0,C 180,E1 -13094.367,E2 -13094.367} C_VEL
LIN {X 0,Y 361.853,Z 494.529,A -85,B 0,C 180,E1 -13097.564,E2 -13097.564} C_VEL
LIN {X 0,Y 361.871,Z 494.53,A -85,B 0,C 180,E1 -13100.971,E2 -13100.971} C_VEL
LIN {X 0,Y 361.87,Z 494.533,A -85,B 0,C 180,E1 -13104.654,E2 -13104.654} C_VEL
LIN {X 0,Y 361.833,Z 494.532,A -85,B 0,C 180,E1 -13108.37,E2 -13108.37} C_VEL
LIN {X 0,Y 361.903,Z 494.514,A -85,B 0,C 180,E1 -13112.22,E2 -13112.22} C_VEL
LIN {X 0,Y 361.921,Z 494.521,A -85,B 0,C 180,E1 -13114.709,E2 -13114.709} C_VEL
LIN {X 0,Y 361.856,Z 494.522,A -85,B 0,C 180,E1 -13118.344,E2 -13118.344} C_VEL
LIN {X 0,Y 361.961,Z 494.521,A -85,B 0,C 180,E1 -13122.061,E2 -13122.061} C_VEL
LIN {X 0,Y 361.991,Z 494.493,A -85,B 0,C 180,E1 -13126.101,E2 -13126.101} C_VEL
LIN {X 0,Y 362.024,Z 494.514,A -85,B 0,C 180,E1 -13129.937,E2 -13129.937} C_VEL
LIN {X 0,Y 362.157,Z 494.476,A -85,B 0,C 180,E1 -13133.313,E2 -13133.313} C_VEL
LIN {X 0,Y 362.275,Z 494.482,A -85,B 0,C 180,E1 -13137.776,E2 -13137.776} C_VEL
LIN {X 0,Y 362.419,Z 494.453,A -85,B 0,C 180,E1 -13139.999,E2 -13139.999} C_VEL
LIN {X 0,Y 362.275,Z 494.456,A -85,B 0,C 180,E1 -13142.223,E2 -13142.223} C_VEL
LIN {X 0,Y 362.154,Z 494.494,A -85,B 0,C 180,E1 -13146.686,E2 -13146.686} C_VEL
LIN {X 0,Y 362.023,Z 494.491,A -85,B 0,C 180,E1 -13150.062,E2 -13150.062} C_VEL
LIN {X 0,Y 361.989,Z 494.519,A -85,B 0,C 180,E1 -13153.898,E2 -13153.898} C_VEL
LIN {X 0,Y 361.959,Z 494.503,A -85,B 0,C 180,E1 -13157.938,E2 -13157.938} C_VEL
LIN {X 0,Y 361.885,Z 494.531,A -85,B 0,C 180,E1 -13161.653,E2 -13161.653} C_VEL
LIN {X 0,Y 361.92,Z 494.512,A -85,B 0,C 180,E1 -13165.29,E2 -13165.29} C_VEL
LIN {X 0,Y 361.914,Z 494.529,A -85,B 0,C 180,E1 -13167.778,E2 -13167.778} C_VEL
LIN {X 0,Y 361.851,Z 494.524,A -85,B 0,C 180,E1 -13171.627,E2 -13171.627} C_VEL
LIN {X 0,Y 361.867,Z 494.524,A -85,B 0,C 180,E1 -13175.345,E2 -13175.345} C_VEL
LIN {X 0,Y 361.865,Z 494.534,A -85,B 0,C 180,E1 -13179.027,E2 -13179.027} C_VEL
LIN {X 0,Y 361.885,Z 494.532,A -85,B 0,C 180,E1 -13182.442,E2 -13182.442} C_VEL
LIN {X 0,Y 361.922,Z 494.491,A -85,B 0,C 180,E1 -13185.929,E2 -13185.929} C_VEL
LIN {X 0,Y 361.899,Z 494.524,A -85,B 0,C 180,E1 -13189.232,E2 -13189.232} C_VEL
LIN {X 0,Y 361.863,Z 494.508,A -85,B 0,C 180,E1 -13192.983,E2 -13192.983} C_VEL
LIN {X 0,Y 361.854,Z 494.537,A -85,B 0,C 180,E1 -13196.63,E2 -13196.63} C_VEL
LIN {X 0,Y 361.871,Z 494.537,A -85,B 0,C 180,E1 -13199.673,E2 -13199.673} C_VEL
LIN {X 0,Y 361.95,Z 494.526,A -85,B 0,C 180,E1 -13203.475,E2 -13203.475} C_VEL
LIN {X 0,Y 361.885,Z 494.534,A -85,B 0,C 180,E1 -13207.145,E2 -13207.145} C_VEL
LIN {X 0,Y 361.939,Z 494.81,A -85,B 0,C 180,E1 -13209.099,E2 -13209.099} C_VEL
LIN {X 0,Y 362.245,Z 496.005,A -85,B 0,C 180,E1 -13209.442,E2 -13209.442} C_VEL
LIN {X 0,Y 363.608,Z 498.347,A -85,B 0,C 180,E1 -13209.973,E2 -13209.973} C_VEL
LIN {X 0,Y 365.973,Z 500.123,A -85,B 0,C 180,E1 -13210.786,E2 -13210.786} C_VEL
LIN {X 0,Y 366.881,Z 500.824,A -85,B 0,C 180,E1 -13211.104,E2 -13211.104} C_VEL
LIN {X 0,Y 368.719,Z 503.838,A -85,B 0,C 180,E1 -13211.85,E2 -13211.85} C_VEL
LIN {X 0,Y 371.414,Z 505.962,A -85,B 0,C 180,E1 -13212.882,E2 -13212.882} C_VEL
LIN {X 0,Y 372.416,Z 506.713,A -85,B 0,C 180,E1 -13213.275,E2 -13213.275} C_VEL
LIN {X 0,Y 374.492,Z 509.81,A -85,B 0,C 180,E1 -13214.21,E2 -13214.21} C_VEL
LIN {X 0,Y 377.194,Z 511.951,A -85,B 0,C 180,E1 -13215.419,E2 -13215.419} C_VEL
LIN {X 0,Y 378.542,Z 512.798,A -85,B 0,C 180,E1 -13216.034,E2 -13216.034} C_VEL
LIN {X 0,Y 380.543,Z 515.815,A -85,B 0,C 180,E1 -13217.13,E2 -13217.13} C_VEL
LIN {X 0,Y 383.157,Z 517.993,A -85,B 0,C 180,E1 -13218.585,E2 -13218.585} C_VEL
LIN {X 0,Y 385.31,Z 519.126,A -85,B 0,C 180,E1 -13219.889,E2 -13219.889} C_VEL
LIN {X 0,Y 386.903,Z 521.497,A -85,B 0,C 180,E1 -13221.118,E2 -13221.118} C_VEL
LIN {X 0,Y 388.554,Z 523.28,A -85,B 0,C 180,E1 -13222.501,E2 -13222.501} C_VEL
LIN {X 0,Y 390.571,Z 524.66,A -85,B 0,C 180,E1 -13224.579,E2 -13224.579} C_VEL
LIN {X 0,Y 391.514,Z 525.139,A -85,B 0,C 180,E1 -13225.883,E2 -13225.883} C_VEL
LIN {X 0,Y 392.525,Z 525.53,A -85,B 0,C 180,E1 -13227.948,E2 -13227.948} C_VEL
LIN {X 0,Y 392.765,Z 525.737,A -85,B 0,C 180,E1 -13228.975,E2 -13228.975} C_VEL
LIN {X 0,Y 392.765,Z 525.74,A -85,B 0,C 180,E1 -13231.025,E2 -13231.025} C_VEL
LIN {X 0,Y 392.117,Z 525.257,A -85,B 0,C 180,E1 -13233.082,E2 -13233.082} C_VEL
LIN {X 0,Y 390.773,Z 524.769,A -85,B 0,C 180,E1 -13235.159,E2 -13235.159} C_VEL
LIN {X 0,Y 388.801,Z 523.472,A -85,B 0,C 180,E1 -13237.269,E2 -13237.269} C_VEL
LIN {X 0,Y 386.986,Z 521.604,A -85,B 0,C 180,E1 -13238.815,E2 -13238.815} C_VEL
LIN {X 0,Y 385.11,Z 518.919,A -85,B 0,C 180,E1 -13240.249,E2 -13240.249} C_VEL
LIN {X 0,Y 382.116,Z 517.268,A -85,B 0,C 180,E1 -13242.009,E2 -13242.009} C_VEL
LIN {X 0,Y 379.62,Z 514.647,A -85,B 0,C 180,E1 -13243.368,E2 -13243.368} C_VEL
LIN {X 0,Y 378.237,Z 512.477,A -85,B 0,C 180,E1 -13244.115,E2 -13244.115} C_VEL
LIN {X 0,Y 375.346,Z 510.626,A -85,B 0,C 180,E1 -13245.405,E2 -13245.405} C_VEL
LIN {X 0,Y 373.172,Z 508.099,A -85,B 0,C 180,E1 -13246.37,E2 -13246.37} C_VEL
LIN {X 0,Y 372.185,Z 506.35,A -85,B 0,C 180,E1 -13246.83,E2 -13246.83} C_VEL
LIN {X 0,Y 369.2,Z 504.338,A -85,B 0,C 180,E1 -13247.969,E2 -13247.969} C_VEL
LIN {X 0,Y 367.352,Z 501.74,A -85,B 0,C 180,E1 -13248.708,E2 -13248.708} C_VEL
LIN {X 0,Y 366.54,Z 500.38,A -85,B 0,C 180,E1 -13249.023,E2 -13249.023} C_VEL
LIN {X 0,Y 363.862,Z 498.621,A -85,B 0,C 180,E1 -13249.94,E2 -13249.94} C_VEL
LIN {X 0,Y 362.292,Z 496.203,A -85,B 0,C 180,E1 -13250.532,E2 -13250.532} C_VEL
LIN {X 0,Y 361.945,Z 494.866,A -85,B 0,C 180,E1 -13250.87,E2 -13250.87} C_VEL
LIN {X 0,Y 361.887,Z 494.534,A -85,B 0,C 180,E1 -13251.653,E2 -13251.653} C_VEL
LIN {X 0,Y 361.923,Z 494.53,A -85,B 0,C 180,E1 -13255.29,E2 -13255.29} C_VEL
LIN {X 0,Y 361.917,Z 494.53,A -85,B 0,C 180,E1 -13257.778,E2 -13257.778} C_VEL
LIN {X 0,Y 361.841,Z 494.538,A -85,B 0,C 180,E1 -13261.285,E2 -13261.285} C_VEL
LIN {X 0,Y 361.849,Z 494.538,A -85,B 0,C 180,E1 -13264.28,E2 -13264.28} C_VEL
LIN {X 0,Y 361.859,Z 494.509,A -85,B 0,C 180,E1 -13267.223,E2 -13267.223} C_VEL
LIN {X 0,Y 361.899,Z 494.524,A -85,B 0,C 180,E1 -13270.768,E2 -13270.768} C_VEL
LIN {X 0,Y 361.925,Z 494.495,A -85,B 0,C 180,E1 -13274.35,E2 -13274.35} C_VEL
LIN {X 0,Y 361.885,Z 494.532,A -85,B 0,C 180,E1 -13277.558,E2 -13277.558} C_VEL
LIN {X 0,Y 361.877,Z 494.521,A -85,B 0,C 180,E1 -13279.609,E2 -13279.609} C_VEL
LIN {X 0,Y 361.194,Z 494.616,A -85,B 0,C 180,E1 -13280.538,E2 -13280.538} C_VEL
LIN {X 0,Y 358.342,Z 494.975,A -85,B 0,C 180,E1 -13282.047,E2 -13282.047} C_VEL
LIN {X 0,Y 355.932,Z 495.266,A -85,B 0,C 180,E1 -13283.269,E2 -13283.269} C_VEL
LIN {X 0,Y 354.893,Z 495.39,A -85,B 0,C 180,E1 -13284.214,E2 -13284.214} C_VEL
LIN {X 0,Y 354.806,Z 495.403,A -85,B 0,C 180,E1 -13284.534,E2 -13284.534} C_VEL
LIN {X 0,Y 354.79,Z 495.414,A -85,B 0,C 180,E1 -13287.668,E2 -13287.668} C_VEL
LIN {X 0,Y 354.861,Z 495.396,A -85,B 0,C 180,E1 -13290.621,E2 -13290.621} C_VEL
LIN {X 0,Y 354.891,Z 495.393,A -85,B 0,C 180,E1 -13294.173,E2 -13294.173} C_VEL
LIN {X 0,Y 354.828,Z 495.405,A -85,B 0,C 180,E1 -13297.894,E2 -13297.894} C_VEL
LIN {X 0,Y 354.914,Z 495.381,A -85,B 0,C 180,E1 -13301.892,E2 -13301.892} C_VEL
LIN {X 0,Y 354.934,Z 495.397,A -85,B 0,C 180,E1 -13305.982,E2 -13305.982} C_VEL
LIN {X 0,Y 354.97,Z 495.369,A -85,B 0,C 180,E1 -13309.736,E2 -13309.736} C_VEL
LIN {X 0,Y 355.121,Z 495.371,A -85,B 0,C 180,E1 -13313.181,E2 -13313.181} C_VEL
LIN {X 0,Y 355.238,Z 495.331,A -85,B 0,C 180,E1 -13317.733,E2 -13317.733} C_VEL
LIN {X 0,Y 355.389,Z 495.329,A -85,B 0,C 180,E1 -13320.001,E2 -13320.001} C_VEL
LIN {X 0,Y 355.238,Z 495.359,A -85,B 0,C 180,E1 -13322.268,E2 -13322.268} C_VEL
LIN {X 0,Y 355.121,Z 495.354,A -85,B 0,C 180,E1 -13326.82,E2 -13326.82} C_VEL
LIN {X 0,Y 354.971,Z 495.395,A -85,B 0,C 180,E1 -13330.265,E2 -13330.265} C_VEL
LIN {X 0,Y 354.936,Z 495.372,A -85,B 0,C 180,E1 -13334.019,E2 -13334.019} C_VEL
LIN {X 0,Y 354.916,Z 495.399,A -85,B 0,C 180,E1 -13338.109,E2 -13338.109} C_VEL
LIN {X 0,Y 354.811,Z 495.401,A -85,B 0,C 180,E1 -13342.108,E2 -13342.108} C_VEL
LIN {X 0,Y 354.893,Z 495.396,A -85,B 0,C 180,E1 -13345.828,E2 -13345.828} C_VEL
LIN {X 0,Y 354.813,Z 495.411,A -85,B 0,C 180,E1 -13349.683,E2 -13349.683} C_VEL
LIN {X 0,Y 354.802,Z 495.402,A -85,B 0,C 180,E1 -13353.703,E2 -13353.703} C_VEL
LIN {X 0,Y 354.796,Z 495.415,A -85,B 0,C 180,E1 -13356.46,E2 -13356.46} C_VEL
LIN {X 0,Y 354.821,Z 495.412,A -85,B 0,C 180,E1 -13359.425,E2 -13359.425} C_VEL
LIN {X 0,Y 354.801,Z 495.412,A -85,B 0,C 180,E1 -13362.871,E2 -13362.871} C_VEL
LIN {X 0,Y 354.765,Z 495.397,A -85,B 0,C 180,E1 -13366.105,E2 -13366.105} C_VEL
LIN {X 0,Y 354.787,Z 495.418,A -85,B 0,C 180,E1 -13369.18,E2 -13369.18} C_VEL
LIN {X 0,Y 354.806,Z 495.351,A -85,B 0,C 180,E1 -13372.403,E2 -13372.403} C_VEL
LIN {X 0,Y 354.876,Z 495.503,A -85,B 0,C 180,E1 -13374.949,E2 -13374.949} C_VEL
LIN {X 0,Y 356.34,Z 502.154,A -85,B 0,C 180,E1 -13377.156,E2 -13377.156} C_VEL
LIN {X 0,Y 358.428,Z 512.223,A -85,B 0,C 180,E1 -13380.192,E2 -13380.192} C_VEL
LIN {X 0,Y 359.514,Z 518.293,A -85,B 0,C 180,E1 -13382.02,E2 -13382.02} C_VEL
LIN {X 0,Y 359.489,Z 520.575,A -85,B 0,C 180,E1 -13382.596,E2 -13382.596} C_VEL
LIN {X 0,Y 364.387,Z 541.78,A -85,B 0,C 180,E1 -13383.486,E2 -13383.486} C_VEL
LIN {X 0,Y 368.356,Z 562.81,A -85,B 0,C 180,E1 -13384.237,E2 -13384.237} C_VEL
LIN {X 0,Y 366.29,Z 654.736,A -85,B 0,C 180,E1 -13386.052,E2 -13386.052} C_VEL
LIN {X 0,Y 365.717,Z 666.092,A -85,B 0,C 180,E1 -13386.388,E2 -13386.388} C_VEL
LIN {X 0,Y 364.963,Z 676.633,A -85,B 0,C 180,E1 -13386.824,E2 -13386.824} C_VEL
LIN {X 0,Y 364.017,Z 687.787,A -85,B 0,C 180,E1 -13387.436,E2 -13387.436} C_VEL
LIN {X 0,Y 363.088,Z 697.76,A -85,B 0,C 180,E1 -13388.124,E2 -13388.124} C_VEL
LIN {X 0,Y 362.166,Z 706.41,A -85,B 0,C 180,E1 -13388.832,E2 -13388.832} C_VEL
LIN {X 0,Y 360.786,Z 717.407,A -85,B 0,C 180,E1 -13389.921,E2 -13389.921} C_VEL
LIN {X 0,Y 359.483,Z 726.826,A -85,B 0,C 180,E1 -13391.033,E2 -13391.033} C_VEL
LIN {X 0,Y 358.247,Z 735.849,A -85,B 0,C 180,E1 -13392.298,E2 -13392.298} C_VEL
LIN {X 0,Y 357.259,Z 742.824,A -85,B 0,C 180,E1 -13393.427,E2 -13393.427} C_VEL
LIN {X 0,Y 356.248,Z 750.35,A -85,B 0,C 180,E1 -13394.848,E2 -13394.848} C_VEL
LIN {X 0,Y 355.466,Z 756.829,A -85,B 0,C 180,E1 -13396.276,E2 -13396.276} C_VEL
LIN {X 0,Y 354.652,Z 763.371,A -85,B 0,C 180,E1 -13397.991,E2 -13397.991} C_VEL
LIN {X 0,Y 354,Z 768.803,A -85,B 0,C 180,E1 -13399.707,E2 -13399.707} C_VEL
LIN {X 0,Y 353.61,Z 773.249,A -85,B 0,C 180,E1 -13401.428,E2 -13401.428} C_VEL
LIN {X 0,Y 353.397,Z 776.795,A -85,B 0,C 180,E1 -13403.147,E2 -13403.147} C_VEL
LIN {X 0,Y 353.282,Z 778.734,A -85,B 0,C 180,E1 -13404.292,E2 -13404.292} C_VEL
LIN {X 0,Y 353.212,Z 781.418,A -85,B 0,C 180,E1 -13406.578,E2 -13406.578} C_VEL
LIN {X 0,Y 353.215,Z 782.708,A -85,B 0,C 180,E1 -13408.86,E2 -13408.86} C_VEL
LIN {X 0,Y 353.261,Z 782.961,A -85,B 0,C 180,E1 -13410,E2 -13410} C_VEL
LIN {X 0,Y 353.17,Z 782.234,A -85,B 0,C 180,E1 -13412.281,E2 -13412.281} C_VEL
LIN {X 0,Y 353.212,Z 781.418,A -85,B 0,C 180,E1 -13413.422,E2 -13413.422} C_VEL
LIN {X 0,Y 353.315,Z 778.299,A -85,B 0,C 180,E1 -13415.965,E2 -13415.965} C_VEL
LIN {X 0,Y 353.519,Z 774.516,A -85,B 0,C 180,E1 -13417.999,E2 -13417.999} C_VEL
LIN {X 0,Y 353.843,Z 770.382,A -85,B 0,C 180,E1 -13419.719,E2 -13419.719} C_VEL
LIN {X 0,Y 354.356,Z 765.282,A -85,B 0,C 180,E1 -13421.439,E2 -13421.439} C_VEL
LIN {X 0,Y 355.062,Z 760.244,A -85,B 0,C 180,E1 -13422.866,E2 -13422.866} C_VEL
LIN {X 0,Y 355.752,Z 754.138,A -85,B 0,C 180,E1 -13424.346,E2 -13424.346} C_VEL
LIN {X 0,Y 356.828,Z 745.949,A -85,B 0,C 180,E1 -13426.006,E2 -13426.006} C_VEL
LIN {X 0,Y 357.727,Z 739.486,A -85,B 0,C 180,E1 -13427.139,E2 -13427.139} C_VEL
LIN {X 0,Y 359.042,Z 730.005,A -85,B 0,C 180,E1 -13428.547,E2 -13428.547} C_VEL
LIN {X 0,Y 360.321,Z 721.129,A -85,B 0,C 180,E1 -13429.661,E2 -13429.661} C_VEL
LIN {X 0,Y 361.588,Z 711.454,A -85,B 0,C 180,E1 -13430.69,E2 -13430.69} C_VEL
LIN {X 0,Y 362.683,Z 701.267,A -85,B 0,C 180,E1 -13431.603,E2 -13431.603} C_VEL
LIN {X 0,Y 363.732,Z 691.008,A -85,B 0,C 180,E1 -13432.358,E2 -13432.358} C_VEL
LIN {X 0,Y 364.734,Z 679.353,A -85,B 0,C 180,E1 -13433.041,E2 -13433.041} C_VEL
LIN {X 0,Y 365.604,Z 667.916,A -85,B 0,C 180,E1 -13433.545,E2 -13433.545} C_VEL
LIN {X 0,Y 366.171,Z 657.413,A -85,B 0,C 180,E1 -13433.882,E2 -13433.882} C_VEL
LIN {X 0,Y 367.042,Z 627.304,A -85,B 0,C 180,E1 -13434.498,E2 -13434.498} C_VEL
LIN {X 0,Y 368.265,Z 561.788,A -85,B 0,C 180,E1 -13435.792,E2 -13435.792} C_VEL
LIN {X 0,Y 363.038,Z 535.724,A -85,B 0,C 180,E1 -13436.751,E2 -13436.751} C_VEL
LIN {X 0,Y 359.513,Z 520.546,A -85,B 0,C 180,E1 -13437.404,E2 -13437.404} C_VEL
LIN {X 0,Y 359.525,Z 518.294,A -85,B 0,C 180,E1 -13437.979,E2 -13437.979} C_VEL
LIN {X 0,Y 357.854,Z 509.27,A -85,B 0,C 180,E1 -13440.704,E2 -13440.704} C_VEL
LIN {X 0,Y 355.646,Z 498.917,A -85,B 0,C 180,E1 -13443.903,E2 -13443.903} C_VEL
LIN {X 0,Y 354.876,Z 495.502,A -85,B 0,C 180,E1 -13445.051,E2 -13445.051} C_VEL
LIN {X 0,Y 354.804,Z 495.355,A -85,B 0,C 180,E1 -13447.882,E2 -13447.882} C_VEL
LIN {X 0,Y 354.787,Z 495.414,A -85,B 0,C 180,E1 -13451.171,E2 -13451.171} C_VEL
LIN {X 0,Y 354.762,Z 495.403,A -85,B 0,C 180,E1 -13454.505,E2 -13454.505} C_VEL
LIN {X 0,Y 354.81,Z 495.405,A -85,B 0,C 180,E1 -13457.664,E2 -13457.664} C_VEL
LIN {X 0,Y 354.834,Z 495.41,A -85,B 0,C 180,E1 -13460.668,E2 -13460.668} C_VEL
LIN {X 0,Y 354.818,Z 495.411,A -85,B 0,C 180,E1 -13464.3,E2 -13464.3} C_VEL
LIN {X 0,Y 354.782,Z 495.405,A -85,B 0,C 180,E1 -13467.666,E2 -13467.666} C_VEL
LIN {X 0,Y 354.841,Z 495.397,A -85,B 0,C 180,E1 -13471.618,E2 -13471.618} C_VEL
LIN {X 0,Y 354.893,Z 495.396,A -85,B 0,C 180,E1 -13474.172,E2 -13474.172} C_VEL
LIN {X 0,Y 354.811,Z 495.401,A -85,B 0,C 180,E1 -13477.892,E2 -13477.892} C_VEL
LIN {X 0,Y 354.916,Z 495.399,A -85,B 0,C 180,E1 -13481.891,E2 -13481.891} C_VEL
LIN {X 0,Y 354.936,Z 495.372,A -85,B 0,C 180,E1 -13485.981,E2 -13485.981} C_VEL
LIN {X 0,Y 354.971,Z 495.395,A -85,B 0,C 180,E1 -13489.735,E2 -13489.735} C_VEL
LIN {X 0,Y 355.121,Z 495.354,A -85,B 0,C 180,E1 -13493.18,E2 -13493.18} C_VEL
LIN {X 0,Y 355.238,Z 495.359,A -85,B 0,C 180,E1 -13497.732,E2 -13497.732} C_VEL
LIN {X 0,Y 355.389,Z 495.329,A -85,B 0,C 180,E1 -13499.999,E2 -13499.999} C_VEL
LIN {X 0,Y 355.238,Z 495.332,A -85,B 0,C 180,E1 -13502.267,E2 -13502.267} C_VEL
LIN {X 0,Y 355.118,Z 495.371,A -85,B 0,C 180,E1 -13506.819,E2 -13506.819} C_VEL
LIN {X 0,Y 354.97,Z 495.369,A -85,B 0,C 180,E1 -13510.264,E2 -13510.264} C_VEL
LIN {X 0,Y 354.934,Z 495.397,A -85,B 0,C 180,E1 -13514.018,E2 -13514.018} C_VEL
LIN {X 0,Y 354.914,Z 495.381,A -85,B 0,C 180,E1 -13518.108,E2 -13518.108} C_VEL
LIN {X 0,Y 354.828,Z 495.405,A -85,B 0,C 180,E1 -13522.106,E2 -13522.106} C_VEL
LIN {X 0,Y 354.891,Z 495.393,A -85,B 0,C 180,E1 -13525.827,E2 -13525.827} C_VEL
LIN {X 0,Y 354.847,Z 495.394,A -85,B 0,C 180,E1 -13529.678,E2 -13529.678} C_VEL
LIN {X 0,Y 354.823,Z 495.413,A -85,B 0,C 180,E1 -13533.682,E2 -13533.682} C_VEL
LIN {X 0,Y 354.791,Z 495.404,A -85,B 0,C 180,E1 -13536.459,E2 -13536.459} C_VEL
LIN {X 0,Y 354.817,Z 495.411,A -85,B 0,C 180,E1 -13539.424,E2 -13539.424} C_VEL
LIN {X 0,Y 354.837,Z 495.41,A -85,B 0,C 180,E1 -13542.877,E2 -13542.877} C_VEL
LIN {X 0,Y 354.859,Z 495.368,A -85,B 0,C 180,E1 -13546.119,E2 -13546.119} C_VEL
LIN {X 0,Y 354.85,Z 495.401,A -85,B 0,C 180,E1 -13549.189,E2 -13549.189} C_VEL
LIN {X 0,Y 354.803,Z 495.391,A -85,B 0,C 180,E1 -13552.402,E2 -13552.402} C_VEL
LIN {X 0,Y 354.806,Z 495.404,A -85,B 0,C 180,E1 -13554.941,E2 -13554.941} C_VEL
LIN {X 0,Y 354.788,Z 495.418,A -85,B 0,C 180,E1 -13558.405,E2 -13558.405} C_VEL
LIN {X 0,Y 354.848,Z 495.41,A -85,B 0,C 180,E1 -13561.62,E2 -13561.62} C_VEL
LIN {X 0,Y 354.894,Z 495.404,A -85,B 0,C 180,E1 -13564.173,E2 -13564.173} C_VEL
LIN {X 0,Y 354.885,Z 495.653,A -85,B 0,C 180,E1 -13567.134,E2 -13567.134} C_VEL
LIN {X 0,Y 355.169,Z 496.794,A -85,B 0,C 180,E1 -13567.468,E2 -13567.468} C_VEL
LIN {X 0,Y 356.44,Z 499.109,A -85,B 0,C 180,E1 -13567.925,E2 -13567.925} C_VEL
LIN {X 0,Y 359.101,Z 501.098,A -85,B 0,C 180,E1 -13568.75,E2 -13568.75} C_VEL
LIN {X 0,Y 361.608,Z 504.814,A -85,B 0,C 180,E1 -13569.635,E2 -13569.635} C_VEL
LIN {X 0,Y 364.538,Z 507.001,A -85,B 0,C 180,E1 -13570.627,E2 -13570.627} C_VEL
LIN {X 0,Y 367.018,Z 510.537,A -85,B 0,C 180,E1 -13571.582,E2 -13571.582} C_VEL
LIN {X 0,Y 369.94,Z 512.789,A -85,B 0,C 180,E1 -13572.684,E2 -13572.684} C_VEL
LIN {X 0,Y 370.834,Z 513.746,A -85,B 0,C 180,E1 -13573.043,E2 -13573.043} C_VEL
LIN {X 0,Y 373.294,Z 516.866,A -85,B 0,C 180,E1 -13574.105,E2 -13574.105} C_VEL
LIN {X 0,Y 376.179,Z 519.01,A -85,B 0,C 180,E1 -13575.379,E2 -13575.379} C_VEL
LIN {X 0,Y 377.106,Z 519.673,A -85,B 0,C 180,E1 -13575.806,E2 -13575.806} C_VEL
LIN {X 0,Y 379.15,Z 522.579,A -85,B 0,C 180,E1 -13576.882,E2 -13576.882} C_VEL
LIN {X 0,Y 381.774,Z 524.786,A -85,B 0,C 180,E1 -13578.317,E2 -13578.317} C_VEL
LIN {X 0,Y 384.216,Z 526.194,A -85,B 0,C 180,E1 -13579.766,E2 -13579.766} C_VEL
LIN {X 0,Y 386.111,Z 528.834,A -85,B 0,C 180,E1 -13581.207,E2 -13581.207} C_VEL
LIN {X 0,Y 388.199,Z 530.776,A -85,B 0,C 180,E1 -13583.004,E2 -13583.004} C_VEL
LIN {X 0,Y 390.091,Z 531.924,A -85,B 0,C 180,E1 -13585.079,E2 -13585.079} C_VEL
LIN {X 0,Y 391.444,Z 532.438,A -85,B 0,C 180,E1 -13587.334,E2 -13587.334} C_VEL
LIN {X 0,Y 391.9,Z 532.783,A -85,B 0,C 180,E1 -13588.972,E2 -13588.972} C_VEL
LIN {X 0,Y 391.9,Z 532.786,A -85,B 0,C 180,E1 -13591.028,E2 -13591.028} C_VEL
LIN {X 0,Y 391.246,Z 532.301,A -85,B 0,C 180,E1 -13593.089,E2 -13593.089} C_VEL
LIN {X 0,Y 389.893,Z 531.815,A -85,B 0,C 180,E1 -13595.171,E2 -13595.171} C_VEL
LIN {X 0,Y 387.905,Z 530.532,A -85,B 0,C 180,E1 -13597.286,E2 -13597.286} C_VEL
LIN {X 0,Y 386.057,Z 528.752,A -85,B 0,C 180,E1 -13598.837,E2 -13598.837} C_VEL
LIN {X 0,Y 383.71,Z 525.765,A -85,B 0,C 180,E1 -13600.554,E2 -13600.554} C_VEL
LIN {X 0,Y 380.616,Z 523.957,A -85,B 0,C 180,E1 -13602.327,E2 -13602.327} C_VEL
LIN {X 0,Y 378.026,Z 521.196,A -85,B 0,C 180,E1 -13603.705,E2 -13603.705} C_VEL
LIN {X 0,Y 376.798,Z 519.323,A -85,B 0,C 180,E1 -13604.342,E2 -13604.342} C_VEL
LIN {X 0,Y 373.774,Z 517.333,A -85,B 0,C 180,E1 -13605.681,E2 -13605.681} C_VEL
LIN {X 0,Y 371.171,Z 514.271,A -85,B 0,C 180,E1 -13606.815,E2 -13606.815} C_VEL
LIN {X 0,Y 370.322,Z 513.004,A -85,B 0,C 180,E1 -13607.171,E2 -13607.171} C_VEL
LIN {X 0,Y 367.238,Z 510.744,A -85,B 0,C 180,E1 -13608.335,E2 -13608.335} C_VEL
LIN {X 0,Y 365.142,Z 507.937,A -85,B 0,C 180,E1 -13609.139,E2 -13609.139} C_VEL
LIN {X 0,Y 364.54,Z 507.004,A -85,B 0,C 180,E1 -13609.373,E2 -13609.373} C_VEL
LIN {X 0,Y 361.609,Z 504.817,A -85,B 0,C 180,E1 -13610.365,E2 -13610.365} C_VEL
LIN {X 0,Y 359.642,Z 501.898,A -85,B 0,C 180,E1 -13611.059,E2 -13611.059} C_VEL
LIN {X 0,Y 359.1,Z 501.1,A -85,B 0,C 180,E1 -13611.25,E2 -13611.25} C_VEL
LIN {X 0,Y 356.44,Z 499.109,A -85,B 0,C 180,E1 -13612.074,E2 -13612.074} C_VEL
LIN {X 0,Y 355.036,Z 496.422,A -85,B 0,C 180,E1 -13612.6,E2 -13612.6} C_VEL
LIN {X 0,Y 354.876,Z 495.547,A -85,B 0,C 180,E1 -13612.947,E2 -13612.947} C_VEL
LIN {X 0,Y 354.894,Z 495.404,A -85,B 0,C 180,E1 -13615.827,E2 -13615.827} C_VEL
LIN {X 0,Y 354.849,Z 495.411,A -85,B 0,C 180,E1 -13619.678,E2 -13619.678} C_VEL
LIN {X 0,Y 354.8,Z 495.417,A -85,B 0,C 180,E1 -13623.702,E2 -13623.702} C_VEL
LIN {X 0,Y 354.793,Z 495.387,A -85,B 0,C 180,E1 -13626.459,E2 -13626.459} C_VEL
LIN {X 0,Y 354.818,Z 495.412,A -85,B 0,C 180,E1 -13629.423,E2 -13629.423} C_VEL
LIN {X 0,Y 354.834,Z 495.368,A -85,B 0,C 180,E1 -13632.876,E2 -13632.876} C_VEL
LIN {X 0,Y 354.861,Z 495.403,A -85,B 0,C 180,E1 -13636.119,E2 -13636.119} C_VEL
LIN {X 0,Y 354.818,Z 495.4,A -85,B 0,C 180,E1 -13639.599,E2 -13639.599} C_VEL
LIN {X 0,Y 354.791,Z 495.404,A -85,B 0,C 180,E1 -13643.541,E2 -13643.541} C_VEL
LIN {X 0,Y 354.806,Z 495.403,A -85,B 0,C 180,E1 -13644.534,E2 -13644.534} C_VEL
LIN {X 0,Y 354.119,Z 495.495,A -85,B 0,C 180,E1 -13645.481,E2 -13645.481} C_VEL
LIN {X 0,Y 351.23,Z 495.857,A -85,B 0,C 180,E1 -13647.021,E2 -13647.021} C_VEL
LIN {X 0,Y 348.817,Z 496.149,A -85,B 0,C 180,E1 -13648.267,E2 -13648.267} C_VEL
LIN {X 0,Y 347.818,Z 496.265,A -85,B 0,C 180,E1 -13649.232,E2 -13649.232} C_VEL
LIN {X 0,Y 347.756,Z 496.272,A -85,B 0,C 180,E1 -13649.559,E2 -13649.559} C_VEL
LIN {X 0,Y 347.845,Z 496.28,A -85,B 0,C 180,E1 -13652.745,E2 -13652.745} C_VEL
LIN {X 0,Y 347.78,Z 496.268,A -85,B 0,C 180,E1 -13656.162,E2 -13656.162} C_VEL
LIN {X 0,Y 347.806,Z 496.285,A -85,B 0,C 180,E1 -13659.91,E2 -13659.91} C_VEL
LIN {X 0,Y 347.858,Z 496.257,A -85,B 0,C 180,E1 -13662.359,E2 -13662.359} C_VEL
LIN {X 0,Y 347.89,Z 496.274,A -85,B 0,C 180,E1 -13665.971,E2 -13665.971} C_VEL
LIN {X 0,Y 347.92,Z 496.248,A -85,B 0,C 180,E1 -13669.526,E2 -13669.526} C_VEL
LIN {X 0,Y 348.086,Z 496.248,A -85,B 0,C 180,E1 -13673.043,E2 -13673.043} C_VEL
LIN {X 0,Y 348.201,Z 496.207,A -85,B 0,C 180,E1 -13677.687,E2 -13677.687} C_VEL
LIN {X 0,Y 348.338,Z 496.207,A -85,B 0,C 180,E1 -13680.001,E2 -13680.001} C_VEL
LIN {X 0,Y 348.201,Z 496.237,A -85,B 0,C 180,E1 -13682.314,E2 -13682.314} C_VEL
LIN {X 0,Y 348.087,Z 496.231,A -85,B 0,C 180,E1 -13686.959,E2 -13686.959} C_VEL
LIN {X 0,Y 347.921,Z 496.271,A -85,B 0,C 180,E1 -13690.475,E2 -13690.475} C_VEL
LIN {X 0,Y 347.892,Z 496.25,A -85,B 0,C 180,E1 -13694.151,E2 -13694.151} C_VEL
LIN {X 0,Y 347.885,Z 496.273,A -85,B 0,C 180,E1 -13698.291,E2 -13698.291} C_VEL
LIN {X 0,Y 347.762,Z 496.276,A -85,B 0,C 180,E1 -13701.627,E2 -13701.627} C_VEL
LIN {X 0,Y 347.806,Z 496.28,A -85,B 0,C 180,E1 -13705.109,E2 -13705.109} C_VEL
LIN {X 0,Y 347.803,Z 496.268,A -85,B 0,C 180,E1 -13707.695,E2 -13707.695} C_VEL
LIN {X 0,Y 347.744,Z 496.294,A -85,B 0,C 180,E1 -13710.349,E2 -13710.349} C_VEL
LIN {X 0,Y 347.744,Z 496.283,A -85,B 0,C 180,E1 -13714.045,E2 -13714.045} C_VEL
LIN {X 0,Y 347.76,Z 496.282,A -85,B 0,C 180,E1 -13717.322,E2 -13717.322} C_VEL
LIN {X 0,Y 347.752,Z 496.295,A -85,B 0,C 180,E1 -13720.295,E2 -13720.295} C_VEL
LIN {X 0,Y 347.741,Z 496.296,A -85,B 0,C 180,E1 -13723.406,E2 -13723.406} C_VEL
LIN {X 0,Y 347.723,Z 496.27,A -85,B 0,C 180,E1 -13726.687,E2 -13726.687} C_VEL
LIN {X 0,Y 347.746,Z 496.285,A -85,B 0,C 180,E1 -13730.174,E2 -13730.174} C_VEL
LIN {X 0,Y 347.76,Z 496.223,A -85,B 0,C 180,E1 -13732.68,E2 -13732.68} C_VEL
LIN {X 0,Y 347.802,Z 496.402,A -85,B 0,C 180,E1 -13734.484,E2 -13734.484} C_VEL
LIN {X 0,Y 349.338,Z 503.115,A -85,B 0,C 180,E1 -13736.756,E2 -13736.756} C_VEL
LIN {X 0,Y 351.514,Z 513.586,A -85,B 0,C 180,E1 -13740.011,E2 -13740.011} C_VEL
LIN {X 0,Y 352.674,Z 520.287,A -85,B 0,C 180,E1 -13742.013,E2 -13742.013} C_VEL
LIN {X 0,Y 354.544,Z 527.907,A -85,B 0,C 180,E1 -13742.386,E2 -13742.386} C_VEL
LIN {X 0,Y 359.633,Z 551.248,A -85,B 0,C 180,E1 -13743.318,E2 -13743.318} C_VEL
LIN {X 0,Y 361.957,Z 563.399,A -85,B 0,C 180,E1 -13743.764,E2 -13743.764} C_VEL
LIN {X 0,Y 359.774,Z 655.857,A -85,B 0,C 180,E1 -13745.628,E2 -13745.628} C_VEL
LIN {X 0,Y 359.17,Z 666.806,A -85,B 0,C 180,E1 -13745.969,E2 -13745.969} C_VEL
LIN {X 0,Y 358.344,Z 677.795,A -85,B 0,C 180,E1 -13746.447,E2 -13746.447} C_VEL
LIN {X 0,Y 357.452,Z 687.588,A -85,B 0,C 180,E1 -13746.998,E2 -13746.998} C_VEL
LIN {X 0,Y 356.486,Z 697.561,A -85,B 0,C 180,E1 -13747.697,E2 -13747.697} C_VEL
LIN {X 0,Y 355.398,Z 707.225,A -85,B 0,C 180,E1 -13748.515,E2 -13748.515} C_VEL
LIN {X 0,Y 354.105,Z 717.208,A -85,B 0,C 180,E1 -13749.525,E2 -13749.525} C_VEL
LIN {X 0,Y 352.724,Z 726.626,A -85,B 0,C 180,E1 -13750.656,E2 -13750.656} C_VEL
LIN {X 0,Y 351.436,Z 735.649,A -85,B 0,C 180,E1 -13751.943,E2 -13751.943} C_VEL
LIN {X 0,Y 350.408,Z 742.625,A -85,B 0,C 180,E1 -13753.093,E2 -13753.093} C_VEL
LIN {X 0,Y 349.33,Z 750.15,A -85,B 0,C 180,E1 -13754.54,E2 -13754.54} C_VEL
LIN {X 0,Y 348.53,Z 756.629,A -85,B 0,C 180,E1 -13755.997,E2 -13755.997} C_VEL
LIN {X 0,Y 347.655,Z 763.171,A -85,B 0,C 180,E1 -13757.745,E2 -13757.745} C_VEL
LIN {X 0,Y 346.95,Z 768.603,A -85,B 0,C 180,E1 -13759.496,E2 -13759.496} C_VEL
LIN {X 0,Y 346.54,Z 773.049,A -85,B 0,C 180,E1 -13761.251,E2 -13761.251} C_VEL
LIN {X 0,Y 346.322,Z 776.596,A -85,B 0,C 180,E1 -13763.007,E2 -13763.007} C_VEL
LIN {X 0,Y 346.202,Z 778.536,A -85,B 0,C 180,E1 -13764.174,E2 -13764.174} C_VEL
LIN {X 0,Y 346.135,Z 781.221,A -85,B 0,C 180,E1 -13766.508,E2 -13766.508} C_VEL
LIN {X 0,Y 346.115,Z 782.51,A -85,B 0,C 180,E1 -13768.837,E2 -13768.837} C_VEL
LIN {X 0,Y 346.164,Z 782.763,A -85,B 0,C 180,E1 -13770,E2 -13770} C_VEL
LIN {X 0,Y 346.081,Z 782.036,A -85,B 0,C 180,E1 -13772.328,E2 -13772.328} C_VEL
LIN {X 0,Y 346.135,Z 781.221,A -85,B 0,C 180,E1 -13773.492,E2 -13773.492} C_VEL
LIN {X 0,Y 346.235,Z 778.34,A -85,B 0,C 180,E1 -13775.943,E2 -13775.943} C_VEL
LIN {X 0,Y 346.468,Z 774.317,A -85,B 0,C 180,E1 -13778.163,E2 -13778.163} C_VEL
LIN {X 0,Y 346.808,Z 770.183,A -85,B 0,C 180,E1 -13779.918,E2 -13779.918} C_VEL
LIN {X 0,Y 347.37,Z 765.083,A -85,B 0,C 180,E1 -13781.672,E2 -13781.672} C_VEL
LIN {X 0,Y 348.074,Z 760.044,A -85,B 0,C 180,E1 -13783.129,E2 -13783.129} C_VEL
LIN {X 0,Y 348.815,Z 753.507,A -85,B 0,C 180,E1 -13784.733,E2 -13784.733} C_VEL
LIN {X 0,Y 349.957,Z 745.75,A -85,B 0,C 180,E1 -13786.329,E2 -13786.329} C_VEL
LIN {X 0,Y 351.176,Z 737.468,A -85,B 0,C 180,E1 -13787.769,E2 -13787.769} C_VEL
LIN {X 0,Y 352.415,Z 728.745,A -85,B 0,C 180,E1 -13789.059,E2 -13789.059} C_VEL
LIN {X 0,Y 353.792,Z 719.69,A -85,B 0,C 180,E1 -13790.19,E2 -13790.19} C_VEL
LIN {X 0,Y 354.916,Z 711.479,A -85,B 0,C 180,E1 -13791.074,E2 -13791.074} C_VEL
LIN {X 0,Y 356.073,Z 701.069,A -85,B 0,C 180,E1 -13792.025,E2 -13792.025} C_VEL
LIN {X 0,Y 357.174,Z 690.81,A -85,B 0,C 180,E1 -13792.791,E2 -13792.791} C_VEL
LIN {X 0,Y 358.091,Z 680.515,A -85,B 0,C 180,E1 -13793.417,E2 -13793.417} C_VEL
LIN {X 0,Y 359.056,Z 668.63,A -85,B 0,C 180,E1 -13793.963,E2 -13793.963} C_VEL
LIN {X 0,Y 359.682,Z 657.215,A -85,B 0,C 180,E1 -13794.34,E2 -13794.34} C_VEL
LIN {X 0,Y 360.527,Z 628.895,A -85,B 0,C 180,E1 -13794.932,E2 -13794.932} C_VEL
LIN {X 0,Y 361.883,Z 562.83,A -85,B 0,C 180,E1 -13796.254,E2 -13796.254} C_VEL
LIN {X 0,Y 356.943,Z 538.113,A -85,B 0,C 180,E1 -13797.188,E2 -13797.188} C_VEL
LIN {X 0,Y 352.73,Z 520.574,A -85,B 0,C 180,E1 -13797.953,E2 -13797.953} C_VEL
LIN {X 0,Y 352.533,Z 519.111,A -85,B 0,C 180,E1 -13798.274,E2 -13798.274} C_VEL
LIN {X 0,Y 350.64,Z 509.047,A -85,B 0,C 180,E1 -13801.407,E2 -13801.407} C_VEL
LIN {X 0,Y 348.059,Z 497.412,A -85,B 0,C 180,E1 -13805.132,E2 -13805.132} C_VEL
LIN {X 0,Y 347.803,Z 496.41,A -85,B 0,C 180,E1 -13805.516,E2 -13805.516} C_VEL
LIN {X 0,Y 347.751,Z 496.253,A -85,B 0,C 180,E1 -13808.792,E2 -13808.792} C_VEL
LIN {X 0,Y 347.749,Z 496.28,A -85,B 0,C 180,E1 -13811.829,E2 -13811.829} C_VEL
LIN {X 0,Y 347.706,Z 496.288,A -85,B 0,C 180,E1 -13815.025,E2 -13815.025} C_VEL
LIN {X 0,Y 347.765,Z 496.283,A -85,B 0,C 180,E1 -13818.393,E2 -13818.393} C_VEL
LIN {X 0,Y 347.773,Z 496.278,A -85,B 0,C 180,E1 -13822.01,E2 -13822.01} C_VEL
LIN {X 0,Y 347.741,Z 496.286,A -85,B 0,C 180,E1 -13825.535,E2 -13825.535} C_VEL
LIN {X 0,Y 347.74,Z 496.288,A -85,B 0,C 180,E1 -13828.299,E2 -13828.299} C_VEL
LIN {X 0,Y 347.774,Z 496.285,A -85,B 0,C 180,E1 -13830.987,E2 -13830.987} C_VEL
LIN {X 0,Y 347.825,Z 496.268,A -85,B 0,C 180,E1 -13833.607,E2 -13833.607} C_VEL
LIN {X 0,Y 347.78,Z 496.287,A -85,B 0,C 180,E1 -13836.161,E2 -13836.161} C_VEL
LIN {X 0,Y 347.8,Z 496.267,A -85,B 0,C 180,E1 -13839.908,E2 -13839.908} C_VEL
LIN {X 0,Y 347.86,Z 496.276,A -85,B 0,C 180,E1 -13842.358,E2 -13842.358} C_VEL
LIN {X 0,Y 347.891,Z 496.249,A -85,B 0,C 180,E1 -13845.97,E2 -13845.97} C_VEL
LIN {X 0,Y 347.921,Z 496.271,A -85,B 0,C 180,E1 -13849.525,E2 -13849.525} C_VEL
LIN {X 0,Y 348.087,Z 496.231,A -85,B 0,C 180,E1 -13853.041,E2 -13853.041} C_VEL
LIN {X 0,Y 348.201,Z 496.237,A -85,B 0,C 180,E1 -13857.686,E2 -13857.686} C_VEL
LIN {X 0,Y 348.338,Z 496.207,A -85,B 0,C 180,E1 -13859.999,E2 -13859.999} C_VEL
LIN {X 0,Y 348.2,Z 496.207,A -85,B 0,C 180,E1 -13862.313,E2 -13862.313} C_VEL
LIN {X 0,Y 348.084,Z 496.248,A -85,B 0,C 180,E1 -13866.958,E2 -13866.958} C_VEL
LIN {X 0,Y 347.92,Z 496.248,A -85,B 0,C 180,E1 -13870.474,E2 -13870.474} C_VEL
LIN {X 0,Y 347.891,Z 496.273,A -85,B 0,C 180,E1 -13874.15,E2 -13874.15} C_VEL
LIN {X 0,Y 347.883,Z 496.258,A -85,B 0,C 180,E1 -13878.29,E2 -13878.29} C_VEL
LIN {X 0,Y 347.782,Z 496.288,A -85,B 0,C 180,E1 -13881.635,E2 -13881.635} C_VEL
LIN {X 0,Y 347.804,Z 496.268,A -85,B 0,C 180,E1 -13885.108,E2 -13885.108} C_VEL
LIN {X 0,Y 347.804,Z 496.288,A -85,B 0,C 180,E1 -13887.694,E2 -13887.694} C_VEL
LIN {X 0,Y 347.762,Z 496.272,A -85,B 0,C 180,E1 -13890.346,E2 -13890.346} C_VEL
LIN {X 0,Y 347.741,Z 496.291,A -85,B 0,C 180,E1 -13894.044,E2 -13894.044} C_VEL
LIN {X 0,Y 347.755,Z 496.286,A -85,B 0,C 180,E1 -13897.321,E2 -13897.321} C_VEL
LIN {X 0,Y 347.787,Z 496.276,A -85,B 0,C 180,E1 -13900.289,E2 -13900.289} C_VEL
LIN {X 0,Y 347.813,Z 496.288,A -85,B 0,C 180,E1 -13903.393,E2 -13903.393} C_VEL
LIN {X 0,Y 347.81,Z 496.241,A -85,B 0,C 180,E1 -13906.67,E2 -13906.67} C_VEL
LIN {X 0,Y 347.78,Z 496.291,A -85,B 0,C 180,E1 -13910.166,E2 -13910.166} C_VEL
LIN {X 0,Y 347.783,Z 496.264,A -85,B 0,C 180,E1 -13914.125,E2 -13914.125} C_VEL
LIN {X 0,Y 347.734,Z 496.297,A -85,B 0,C 180,E1 -13918.086,E2 -13918.086} C_VEL
LIN {X 0,Y 347.801,Z 496.288,A -85,B 0,C 180,E1 -13920.99,E2 -13920.99} C_VEL
LIN {X 0,Y 347.827,Z 496.285,A -85,B 0,C 180,E1 -13923.608,E2 -13923.608} C_VEL
LIN {X 0,Y 347.836,Z 496.434,A -85,B 0,C 180,E1 -13925.292,E2 -13925.292} C_VEL
LIN {X 0,Y 348.084,Z 497.474,A -85,B 0,C 180,E1 -13925.649,E2 -13925.649} C_VEL
LIN {X 0,Y 349.348,Z 499.923,A -85,B 0,C 180,E1 -13926.083,E2 -13926.083} C_VEL
LIN {X 0,Y 351.789,Z 501.842,A -85,B 0,C 180,E1 -13926.776,E2 -13926.776} C_VEL
LIN {X 0,Y 354.457,Z 505.719,A -85,B 0,C 180,E1 -13927.634,E2 -13927.634} C_VEL
LIN {X 0,Y 357.262,Z 508.063,A -85,B 0,C 180,E1 -13928.503,E2 -13928.503} C_VEL
LIN {X 0,Y 359.704,Z 511.412,A -85,B 0,C 180,E1 -13929.344,E2 -13929.344} C_VEL
LIN {X 0,Y 362.861,Z 514.009,A -85,B 0,C 180,E1 -13930.4,E2 -13930.4} C_VEL
LIN {X 0,Y 365.293,Z 517.201,A -85,B 0,C 180,E1 -13931.31,E2 -13931.31} C_VEL
LIN {X 0,Y 368.904,Z 520.141,A -85,B 0,C 180,E1 -13932.666,E2 -13932.666} C_VEL
LIN {X 0,Y 371.56,Z 523.452,A -85,B 0,C 180,E1 -13933.789,E2 -13933.789} C_VEL
LIN {X 0,Y 374.681,Z 525.748,A -85,B 0,C 180,E1 -13935.116,E2 -13935.116} C_VEL
LIN {X 0,Y 375.732,Z 526.724,A -85,B 0,C 180,E1 -13935.616,E2 -13935.616} C_VEL
LIN {X 0,Y 378.285,Z 529.877,A -85,B 0,C 180,E1 -13936.918,E2 -13936.918} C_VEL
LIN {X 0,Y 381.032,Z 531.951,A -85,B 0,C 180,E1 -13938.408,E2 -13938.408} C_VEL
LIN {X 0,Y 383.008,Z 533.127,A -85,B 0,C 180,E1 -13939.575,E2 -13939.575} C_VEL
LIN {X 0,Y 385.183,Z 535.978,A -85,B 0,C 180,E1 -13941.186,E2 -13941.186} C_VEL
LIN {X 0,Y 387.303,Z 537.831,A -85,B 0,C 180,E1 -13942.988,E2 -13942.988} C_VEL
LIN {X 0,Y 389.213,Z 538.946,A -85,B 0,C 180,E1 -13945.068,E2 -13945.068} C_VEL
LIN {X 0,Y 390.576,Z 539.485,A -85,B 0,C 180,E1 -13947.328,E2 -13947.328} C_VEL
LIN {X 0,Y 391.037,Z 539.805,A -85,B 0,C 180,E1 -13948.97,E2 -13948.97} C_VEL
LIN {X 0,Y 391.037,Z 539.808,A -85,B 0,C 180,E1 -13951.03,E2 -13951.03} C_VEL
LIN {X 0,Y 390.374,Z 539.35,A -85,B 0,C 180,E1 -13953.096,E2 -13953.096} C_VEL
LIN {X 0,Y 389.013,Z 538.856,A -85,B 0,C 180,E1 -13955.183,E2 -13955.183} C_VEL
LIN {X 0,Y 387.01,Z 537.582,A -85,B 0,C 180,E1 -13957.303,E2 -13957.303} C_VEL
LIN {X 0,Y 385.001,Z 535.744,A -85,B 0,C 180,E1 -13958.96,E2 -13958.96} C_VEL
LIN {X 0,Y 382.515,Z 532.679,A -85,B 0,C 180,E1 -13960.734,E2 -13960.734} C_VEL
LIN {X 0,Y 379.401,Z 530.874,A -85,B 0,C 180,E1 -13962.484,E2 -13962.484} C_VEL
LIN {X 0,Y 376.579,Z 527.958,A -85,B 0,C 180,E1 -13963.963,E2 -13963.963} C_VEL
LIN {X 0,Y 375.167,Z 526.064,A -85,B 0,C 180,E1 -13964.661,E2 -13964.661} C_VEL
LIN {X 0,Y 371.759,Z 523.639,A -85,B 0,C 180,E1 -13966.128,E2 -13966.128} C_VEL
LIN {X 0,Y 369.07,Z 520.407,A -85,B 0,C 180,E1 -13967.262,E2 -13967.262} C_VEL
LIN {X 0,Y 368.279,Z 519.517,A -85,B 0,C 180,E1 -13967.587,E2 -13967.587} C_VEL
LIN {X 0,Y 365.055,Z 516.96,A -85,B 0,C 180,E1 -13968.775,E2 -13968.775} C_VEL
LIN {X 0,Y 362.275,Z 513.419,A -85,B 0,C 180,E1 -13969.8,E2 -13969.8} C_VEL
LIN {X 0,Y 359.249,Z 510.941,A -85,B 0,C 180,E1 -13970.806,E2 -13970.806} C_VEL
LIN {X 0,Y 356.803,Z 507.57,A -85,B 0,C 180,E1 -13971.641,E2 -13971.641} C_VEL
LIN {X 0,Y 353.966,Z 505.177,A -85,B 0,C 180,E1 -13972.515,E2 -13972.515} C_VEL
LIN {X 0,Y 351.788,Z 501.846,A -85,B 0,C 180,E1 -13973.224,E2 -13973.224} C_VEL
LIN {X 0,Y 349.348,Z 499.92,A -85,B 0,C 180,E1 -13973.917,E2 -13973.917} C_VEL
LIN {X 0,Y 347.949,Z 496.953,A -85,B 0,C 180,E1 -13974.461,E2 -13974.461} C_VEL
LIN {X 0,Y 347.821,Z 496.365,A -85,B 0,C 180,E1 -13974.789,E2 -13974.789} C_VEL
LIN {X 0,Y 347.807,Z 496.287,A -85,B 0,C 180,E1 -13977.693,E2 -13977.693} C_VEL
LIN {X 0,Y 347.759,Z 496.294,A -85,B 0,C 180,E1 -13980.346,E2 -13980.346} C_VEL
LIN {X 0,Y 347.739,Z 496.293,A -85,B 0,C 180,E1 -13984.464,E2 -13984.464} C_VEL
LIN {X 0,Y 347.77,Z 496.271,A -85,B 0,C 180,E1 -13987.989,E2 -13987.989} C_VEL
LIN {X 0,Y 347.778,Z 496.261,A -85,B 0,C 180,E1 -13991.609,E2 -13991.609} C_VEL
LIN {X 0,Y 347.823,Z 496.263,A -85,B 0,C 180,E1 -13995.006,E2 -13995.006} C_VEL
LIN {X 0,Y 347.779,Z 496.28,A -85,B 0,C 180,E1 -13998.39,E2 -13998.39} C_VEL
LIN {X 0,Y 347.767,Z 496.292,A -85,B 0,C 180,E1 -14002.011,E2 -14002.011} C_VEL
LIN {X 0,Y 347.737,Z 496.289,A -85,B 0,C 180,E1 -14005.536,E2 -14005.536} C_VEL
LIN {X 0,Y 347.756,Z 496.272,A -85,B 0,C 180,E1 -14009.559,E2 -14009.559} C_VEL
LIN {X 0,Y 347.142,Z 496.357,A -85,B 0,C 180,E1 -14010.526,E2 -14010.526} C_VEL
LIN {X 0,Y 344.315,Z 496.72,A -85,B 0,C 180,E1 -14012.101,E2 -14012.101} C_VEL
LIN {X 0,Y 341.887,Z 497.02,A -85,B 0,C 180,E1 -14013.375,E2 -14013.375} C_VEL
LIN {X 0,Y 340.839,Z 497.14,A -85,B 0,C 180,E1 -14014.362,E2 -14014.362} C_VEL
LIN {X 0,Y 340.753,Z 497.147,A -85,B 0,C 180,E1 -14014.696,E2 -14014.696} C_VEL
LIN {X 0,Y 340.733,Z 497.164,A -85,B 0,C 180,E1 -14018.207,E2 -14018.207} C_VEL
LIN {X 0,Y 340.85,Z 497.131,A -85,B 0,C 180,E1 -14021.984,E2 -14021.984} C_VEL
LIN {X 0,Y 340.862,Z 497.148,A -85,B 0,C 180,E1 -14025.705,E2 -14025.705} C_VEL
LIN {X 0,Y 340.863,Z 497.128,A -85,B 0,C 180,E1 -14029.307,E2 -14029.307} C_VEL
LIN {X 0,Y 341.054,Z 497.125,A -85,B 0,C 180,E1 -14032.898,E2 -14032.898} C_VEL
LIN {X 0,Y 341.163,Z 497.083,A -85,B 0,C 180,E1 -14037.639,E2 -14037.639} C_VEL
LIN {X 0,Y 341.288,Z 497.085,A -85,B 0,C 180,E1 -14040.001,E2 -14040.001} C_VEL
LIN {X 0,Y 341.163,Z 497.113,A -85,B 0,C 180,E1 -14042.362,E2 -14042.362} C_VEL
LIN {X 0,Y 341.055,Z 497.109,A -85,B 0,C 180,E1 -14047.103,E2 -14047.103} C_VEL
LIN {X 0,Y 340.864,Z 497.147,A -85,B 0,C 180,E1 -14050.695,E2 -14050.695} C_VEL
LIN {X 0,Y 340.857,Z 497.127,A -85,B 0,C 180,E1 -14054.326,E2 -14054.326} C_VEL
LIN {X 0,Y 340.831,Z 497.149,A -85,B 0,C 180,E1 -14058.467,E2 -14058.467} C_VEL
LIN {X 0,Y 340.712,Z 497.155,A -85,B 0,C 180,E1 -14061.843,E2 -14061.843} C_VEL
LIN {X 0,Y 340.766,Z 497.155,A -85,B 0,C 180,E1 -14065.665,E2 -14065.665} C_VEL
LIN {X 0,Y 340.723,Z 497.154,A -85,B 0,C 180,E1 -14068.322,E2 -14068.322} C_VEL
LIN {X 0,Y 340.693,Z 497.168,A -85,B 0,C 180,E1 -14071.046,E2 -14071.046} C_VEL
LIN {X 0,Y 340.715,Z 497.169,A -85,B 0,C 180,E1 -14075.28,E2 -14075.28} C_VEL
LIN {X 0,Y 340.714,Z 497.159,A -85,B 0,C 180,E1 -14078.389,E2 -14078.389} C_VEL
LIN {X 0,Y 340.728,Z 497.16,A -85,B 0,C 180,E1 -14082.052,E2 -14082.052} C_VEL
LIN {X 0,Y 340.65,Z 497.152,A -85,B 0,C 180,E1 -14086.228,E2 -14086.228} C_VEL
LIN {X 0,Y 340.688,Z 497.173,A -85,B 0,C 180,E1 -14089.754,E2 -14089.754} C_VEL
LIN {X 0,Y 340.704,Z 497.097,A -85,B 0,C 180,E1 -14093.259,E2 -14093.259} C_VEL
LIN {X 0,Y 340.769,Z 497.313,A -85,B 0,C 180,E1 -14094.001,E2 -14094.001} C_VEL
LIN {X 0,Y 342.673,Z 505.727,A -85,B 0,C 180,E1 -14096.865,E2 -14096.865} C_VEL
LIN {X 0,Y 344.692,Z 515.609,A -85,B 0,C 180,E1 -14100.032,E2 -14100.032} C_VEL
LIN {X 0,Y 345.583,Z 520.156,A -85,B 0,C 180,E1 -14101.397,E2 -14101.397} C_VEL
LIN {X 0,Y 347.315,Z 525.466,A -85,B 0,C 180,E1 -14101.71,E2 -14101.71} C_VEL
LIN {X 0,Y 352.216,Z 546.907,A -85,B 0,C 180,E1 -14102.617,E2 -14102.617} C_VEL
LIN {X 0,Y 355.51,Z 564.149,A -85,B 0,C 180,E1 -14103.272,E2 -14103.272} C_VEL
LIN {X 0,Y 353.371,Z 654.354,A -85,B 0,C 180,E1 -14105.118,E2 -14105.118} C_VEL
LIN {X 0,Y 352.78,Z 665.696,A -85,B 0,C 180,E1 -14105.466,E2 -14105.466} C_VEL
LIN {X 0,Y 351.972,Z 676.237,A -85,B 0,C 180,E1 -14105.916,E2 -14105.916} C_VEL
LIN {X 0,Y 350.923,Z 687.39,A -85,B 0,C 180,E1 -14106.545,E2 -14106.545} C_VEL
LIN {X 0,Y 349.904,Z 697.363,A -85,B 0,C 180,E1 -14107.255,E2 -14107.255} C_VEL
LIN {X 0,Y 348.696,Z 707.024,A -85,B 0,C 180,E1 -14108.08,E2 -14108.08} C_VEL
LIN {X 0,Y 347.447,Z 717.01,A -85,B 0,C 180,E1 -14109.114,E2 -14109.114} C_VEL
LIN {X 0,Y 346.005,Z 726.427,A -85,B 0,C 180,E1 -14110.265,E2 -14110.265} C_VEL
LIN {X 0,Y 344.651,Z 735.45,A -85,B 0,C 180,E1 -14111.575,E2 -14111.575} C_VEL
LIN {X 0,Y 343.592,Z 742.426,A -85,B 0,C 180,E1 -14112.748,E2 -14112.748} C_VEL
LIN {X 0,Y 342.435,Z 749.951,A -85,B 0,C 180,E1 -14114.221,E2 -14114.221} C_VEL
LIN {X 0,Y 341.6,Z 756.43,A -85,B 0,C 180,E1 -14115.707,E2 -14115.707} C_VEL
LIN {X 0,Y 340.676,Z 762.972,A -85,B 0,C 180,E1 -14117.49,E2 -14117.49} C_VEL
LIN {X 0,Y 339.911,Z 768.403,A -85,B 0,C 180,E1 -14119.276,E2 -14119.276} C_VEL
LIN {X 0,Y 339.49,Z 772.85,A -85,B 0,C 180,E1 -14121.068,E2 -14121.068} C_VEL
LIN {X 0,Y 339.247,Z 776.397,A -85,B 0,C 180,E1 -14122.86,E2 -14122.86} C_VEL
LIN {X 0,Y 339.111,Z 778.494,A -85,B 0,C 180,E1 -14124.152,E2 -14124.152} C_VEL
LIN {X 0,Y 339.059,Z 781.023,A -85,B 0,C 180,E1 -14126.435,E2 -14126.435} C_VEL
LIN {X 0,Y 339.017,Z 782.312,A -85,B 0,C 180,E1 -14128.812,E2 -14128.812} C_VEL
LIN {X 0,Y 339.066,Z 782.565,A -85,B 0,C 180,E1 -14130,E2 -14130} C_VEL
LIN {X 0,Y 338.996,Z 781.839,A -85,B 0,C 180,E1 -14132.376,E2 -14132.376} C_VEL
LIN {X 0,Y 339.059,Z 781.023,A -85,B 0,C 180,E1 -14133.565,E2 -14133.565} C_VEL
LIN {X 0,Y 339.134,Z 778.338,A -85,B 0,C 180,E1 -14135.947,E2 -14135.947} C_VEL
LIN {X 0,Y 339.323,Z 775.381,A -85,B 0,C 180,E1 -14137.737,E2 -14137.737} C_VEL
LIN {X 0,Y 339.633,Z 771.553,A -85,B 0,C 180,E1 -14139.529,E2 -14139.529} C_VEL
LIN {X 0,Y 340.135,Z 766.788,A -85,B 0,C 180,E1 -14141.32,E2 -14141.32} C_VEL
LIN {X 0,Y 341.076,Z 759.843,A -85,B 0,C 180,E1 -14143.403,E2 -14143.403} C_VEL
LIN {X 0,Y 342.012,Z 752.617,A -85,B 0,C 180,E1 -14145.19,E2 -14145.19} C_VEL
LIN {X 0,Y 343.084,Z 745.55,A -85,B 0,C 180,E1 -14146.665,E2 -14146.665} C_VEL
LIN {X 0,Y 344.377,Z 737.269,A -85,B 0,C 180,E1 -14148.132,E2 -14148.132} C_VEL
LIN {X 0,Y 345.685,Z 728.547,A -85,B 0,C 180,E1 -14149.445,E2 -14149.445} C_VEL
LIN {X 0,Y 347.099,Z 719.49,A -85,B 0,C 180,E1 -14150.597,E2 -14150.597} C_VEL
LIN {X 0,Y 348.439,Z 709.901,A -85,B 0,C 180,E1 -14151.631,E2 -14151.631} C_VEL
LIN {X 0,Y 349.497,Z 700.871,A -85,B 0,C 180,E1 -14152.461,E2 -14152.461} C_VEL
LIN {X 0,Y 350.647,Z 690.612,A -85,B 0,C 180,E1 -14153.24,E2 -14153.24} C_VEL
LIN {X 0,Y 351.601,Z 680.317,A -85,B 0,C 180,E1 -14153.876,E2 -14153.876} C_VEL
LIN {X 0,Y 352.596,Z 668.432,A -85,B 0,C 180,E1 -14154.43,E2 -14154.43} C_VEL
LIN {X 0,Y 353.238,Z 657.017,A -85,B 0,C 180,E1 -14154.814,E2 -14154.814} C_VEL
LIN {X 0,Y 354.168,Z 626.908,A -85,B 0,C 180,E1 -14155.45,E2 -14155.45} C_VEL
LIN {X 0,Y 355.522,Z 563.935,A -85,B 0,C 180,E1 -14156.732,E2 -14156.732} C_VEL
LIN {X 0,Y 350.523,Z 538.881,A -85,B 0,C 180,E1 -14157.706,E2 -14157.706} C_VEL
LIN {X 0,Y 346.569,Z 522.965,A -85,B 0,C 180,E1 -14158.413,E2 -14158.413} C_VEL
LIN {X 0,Y 345.527,Z 519.973,A -85,B 0,C 180,E1 -14158.63,E2 -14158.63} C_VEL
LIN {X 0,Y 343.364,Z 508.82,A -85,B 0,C 180,E1 -14162.151,E2 -14162.151} C_VEL
LIN {X 0,Y 341.008,Z 498.34,A -85,B 0,C 180,E1 -14165.606,E2 -14165.606} C_VEL
LIN {X 0,Y 340.75,Z 497.177,A -85,B 0,C 180,E1 -14166.109,E2 -14166.109} C_VEL
LIN {X 0,Y 340.698,Z 497.16,A -85,B 0,C 180,E1 -14169.752,E2 -14169.752} C_VEL
LIN {X 0,Y 340.674,Z 497.147,A -85,B 0,C 180,E1 -14172.903,E2 -14172.903} C_VEL
LIN {X 0,Y 340.708,Z 497.166,A -85,B 0,C 180,E1 -14177.1,E2 -14177.1} C_VEL
LIN {X 0,Y 340.707,Z 497.169,A -85,B 0,C 180,E1 -14180.248,E2 -14180.248} C_VEL
LIN {X 0,Y 340.707,Z 497.169,A -85,B 0,C 180,E1 -14183.558,E2 -14183.558} C_VEL
LIN {X 0,Y 340.688,Z 497.16,A -85,B 0,C 180,E1 -14186.152,E2 -14186.152} C_VEL
LIN {X 0,Y 340.737,Z 497.164,A -85,B 0,C 180,E1 -14190.328,E2 -14190.328} C_VEL
LIN {X 0,Y 340.798,Z 497.139,A -85,B 0,C 180,E1 -14193.019,E2 -14193.019} C_VEL
LIN {X 0,Y 340.749,Z 497.166,A -85,B 0,C 180,E1 -14195.637,E2 -14195.637} C_VEL
LIN {X 0,Y 340.728,Z 497.145,A -85,B 0,C 180,E1 -14199.472,E2 -14199.472} C_VEL
LIN {X 0,Y 340.852,Z 497.151,A -85,B 0,C 180,E1 -14201.983,E2 -14201.983} C_VEL
LIN {X 0,Y 340.863,Z 497.126,A -85,B 0,C 180,E1 -14205.704,E2 -14205.704} C_VEL
LIN {X 0,Y 340.864,Z 497.147,A -85,B 0,C 180,E1 -14209.305,E2 -14209.305} C_VEL
LIN {X 0,Y 341.055,Z 497.109,A -85,B 0,C 180,E1 -14212.897,E2 -14212.897} C_VEL
LIN {X 0,Y 341.162,Z 497.113,A -85,B 0,C 180,E1 -14217.638,E2 -14217.638} C_VEL
LIN {X 0,Y 341.288,Z 497.085,A -85,B 0,C 180,E1 -14219.999,E2 -14219.999} C_VEL
LIN {X 0,Y 341.162,Z 497.083,A -85,B 0,C 180,E1 -14222.361,E2 -14222.361} C_VEL
LIN {X 0,Y 341.052,Z 497.125,A -85,B 0,C 180,E1 -14227.102,E2 -14227.102} C_VEL
LIN {X 0,Y 340.863,Z 497.128,A -85,B 0,C 180,E1 -14230.693,E2 -14230.693} C_VEL
LIN {X 0,Y 340.855,Z 497.149,A -85,B 0,C 180,E1 -14234.325,E2 -14234.325} C_VEL
LIN {X 0,Y 340.829,Z 497.138,A -85,B 0,C 180,E1 -14238.466,E2 -14238.466} C_VEL
LIN {X 0,Y 340.746,Z 497.161,A -85,B 0,C 180,E1 -14241.857,E2 -14241.857} C_VEL
LIN {X 0,Y 340.765,Z 497.15,A -85,B 0,C 180,E1 -14245.664,E2 -14245.664} C_VEL
LIN {X 0,Y 340.735,Z 497.163,A -85,B 0,C 180,E1 -14248.319,E2 -14248.319} C_VEL
LIN {X 0,Y 340.708,Z 497.152,A -85,B 0,C 180,E1 -14251.043,E2 -14251.043} C_VEL
LIN {X 0,Y 340.71,Z 497.159,A -85,B 0,C 180,E1 -14255.279,E2 -14255.279} C_VEL
LIN {X 0,Y 340.705,Z 497.171,A -85,B 0,C 180,E1 -14258.387,E2 -14258.387} C_VEL
LIN {X 0,Y 340.72,Z 497.156,A -85,B 0,C 180,E1 -14261.304,E2 -14261.304} C_VEL
LIN {X 0,Y 340.774,Z 497.152,A -85,B 0,C 180,E1 -14264.523,E2 -14264.523} C_VEL
LIN {X 0,Y 340.745,Z 497.128,A -85,B 0,C 180,E1 -14267.945,E2 -14267.945} C_VEL
LIN {X 0,Y 340.728,Z 497.169,A -85,B 0,C 180,E1 -14270.253,E2 -14270.253} C_VEL
LIN {X 0,Y 340.705,Z 497.141,A -85,B 0,C 180,E1 -14273.559,E2 -14273.559} C_VEL
